LIN {X 0,Y 405.489,Z 1080.281,A -85,B 0,C 180,E1 13917.147,E2 13917.147} C_VEL
LIN {X 0,Y 408.998,Z 1063.709,A -85,B 0,C 180,E1 13914.736,E2 13914.736} C_VEL
LIN {X 0,Y 412.817,Z 1045.417,A -85,B 0,C 180,E1 13912.472,E2 13912.472} C_VEL
LIN {X 0,Y 416.994,Z 1024.781,A -85,B 0,C 180,E1 13910.291,E2 13910.291} C_VEL
LIN {X 0,Y 420.9,Z 1004.657,A -85,B 0,C 180,E1 13908.488,E2 13908.488} C_VEL
LIN {X 0,Y 424.408,Z 984.623,A -85,B 0,C 180,E1 13906.997,E2 13906.997} C_VEL
LIN {X 0,Y 427.831,Z 963.376,A -85,B 0,C 180,E1 13905.671,E2 13905.671} C_VEL
LIN {X 0,Y 430.64,Z 942.779,A -85,B 0,C 180,E1 13904.632,E2 13904.632} C_VEL
LIN {X 0,Y 433.258,Z 920.08,A -85,B 0,C 180,E1 13903.723,E2 13903.723} C_VEL
LIN {X 0,Y 435.218,Z 898.048,A -85,B 0,C 180,E1 13903.072,E2 13903.072} C_VEL
LIN {X 0,Y 436.86,Z 866.302,A -85,B 0,C 180,E1 13902.413,E2 13902.413} C_VEL
LIN {X 0,Y 445.415,Z 656.553,A -85,B 0,C 180,E1 13898.433,E2 13898.433} C_VEL
LIN {X 0,Y 447.125,Z 611.826,A -85,B 0,C 180,E1 13897.563,E2 13897.563} C_VEL
LIN {X 0,Y 435.207,Z 593.667,A -85,B 0,C 180,E1 13895.175,E2 13895.175} C_VEL
LIN {X 0,Y 424.65,Z 578.968,A -85,B 0,C 180,E1 13892.869,E2 13892.869} C_VEL
LIN {X 0,Y 417.413,Z 569.477,A -85,B 0,C 180,E1 13891.157,E2 13891.157} C_VEL
LIN {X 0,Y 413.791,Z 564.844,A -85,B 0,C 180,E1 13890.252,E2 13890.252} C_VEL
LIN {X 0,Y 409.785,Z 559.833,A -85,B 0,C 180,E1 13889.208,E2 13889.208} C_VEL
LIN {X 0,Y 405.456,Z 554.439,A -85,B 0,C 180,E1 13887.999,E2 13887.999} C_VEL
LIN {X 0,Y 402.661,Z 549.627,A -85,B 0,C 180,E1 13886.548,E2 13886.548} C_VEL
LIN {X 0,Y 400.386,Z 545.696,A -85,B 0,C 180,E1 13885.279,E2 13885.279} C_VEL
LIN {X 0,Y 397.379,Z 541.061,A -85,B 0,C 180,E1 13883.582,E2 13883.582} C_VEL
LIN {X 0,Y 396.535,Z 539.345,A -85,B 0,C 180,E1 13883.006,E2 13883.006} C_VEL
LIN {X 0,Y 394.114,Z 536.079,A -85,B 0,C 180,E1 13881.583,E2 13881.583} C_VEL
LIN {X 0,Y 393.583,Z 534.195,A -85,B 0,C 180,E1 13880.833,E2 13880.833} C_VEL
LIN {X 0,Y 393.553,Z 533.972,A -85,B 0,C 180,E1 13876.835,E2 13876.835} C_VEL
LIN {X 0,Y 393.555,Z 533.997,A -85,B 0,C 180,E1 13872.918,E2 13872.918} C_VEL
LIN {X 0,Y 393.548,Z 533.952,A -85,B 0,C 180,E1 13868.915,E2 13868.915} C_VEL
LIN {X 0,Y 393.557,Z 534.026,A -85,B 0,C 180,E1 13864.955,E2 13864.955} C_VEL
LIN {X 0,Y 393.56,Z 534.017,A -85,B 0,C 180,E1 13860.873,E2 13860.873} C_VEL
LIN {X 0,Y 393.555,Z 534.013,A -85,B 0,C 180,E1 13856.941,E2 13856.941} C_VEL
LIN {X 0,Y 393.549,Z 534.009,A -85,B 0,C 180,E1 13852.995,E2 13852.995} C_VEL
LIN {X 0,Y 393.543,Z 533.975,A -85,B 0,C 180,E1 13849.015,E2 13849.015} C_VEL
LIN {X 0,Y 393.55,Z 533.997,A -85,B 0,C 180,E1 13844.98,E2 13844.98} C_VEL
LIN {X 0,Y 393.552,Z 533.958,A -85,B 0,C 180,E1 13841.022,E2 13841.022} C_VEL
LIN {X 0,Y 393.573,Z 534.093,A -85,B 0,C 180,E1 13836.968,E2 13836.968} C_VEL
LIN {X 0,Y 393.64,Z 534.566,A -85,B 0,C 180,E1 13836.485,E2 13836.485} C_VEL
LIN {X 0,Y 395.297,Z 538.039,A -85,B 0,C 180,E1 13835.173,E2 13835.173} C_VEL
LIN {X 0,Y 396.887,Z 539.799,A -85,B 0,C 180,E1 13834.322,E2 13834.322} C_VEL
LIN {X 0,Y 398.83,Z 543.682,A -85,B 0,C 180,E1 13833.014,E2 13833.014} C_VEL
LIN {X 0,Y 400.178,Z 545.463,A -85,B 0,C 180,E1 13832.307,E2 13832.307} C_VEL
LIN {X 0,Y 402.489,Z 549.53,A -85,B 0,C 180,E1 13830.979,E2 13830.979} C_VEL
LIN {X 0,Y 406.12,Z 555.885,A -85,B 0,C 180,E1 13829.032,E2 13829.032} C_VEL
LIN {X 0,Y 411.461,Z 565.678,A -85,B 0,C 180,E1 13826.355,E2 13826.355} C_VEL
LIN {X 0,Y 417.794,Z 577.852,A -85,B 0,C 180,E1 13823.423,E2 13823.423} C_VEL
LIN {X 0,Y 419.708,Z 581.207,A -85,B 0,C 180,E1 13822.764,E2 13822.764} C_VEL
LIN {X 0,Y 431.985,Z 599.336,A -85,B 0,C 180,E1 13819.994,E2 13819.994} C_VEL
LIN {X 0,Y 441.06,Z 613.989,A -85,B 0,C 180,E1 13818.116,E2 13818.116} C_VEL
LIN {X 0,Y 443.278,Z 632.103,A -85,B 0,C 180,E1 13817.332,E2 13817.332} C_VEL
LIN {X 0,Y 435.43,Z 864.5,A -85,B 0,C 180,E1 13813.233,E2 13813.233} C_VEL
LIN {X 0,Y 434.04,Z 899.876,A -85,B 0,C 180,E1 13812.574,E2 13812.574} C_VEL
LIN {X 0,Y 432.284,Z 921.112,A -85,B 0,C 180,E1 13811.981,E2 13811.981} C_VEL
LIN {X 0,Y 429.933,Z 942.214,A -85,B 0,C 180,E1 13811.159,E2 13811.159} C_VEL
LIN {X 0,Y 427.165,Z 962.307,A -85,B 0,C 180,E1 13810.155,E2 13810.155} C_VEL
LIN {X 0,Y 423.94,Z 981.509,A -85,B 0,C 180,E1 13808.943,E2 13808.943} C_VEL
LIN {X 0,Y 420.069,Z 1001.923,A -85,B 0,C 180,E1 13807.37,E2 13807.37} C_VEL
LIN {X 0,Y 418.412,Z 1010.233,A -85,B 0,C 180,E1 13806.635,E2 13806.635} C_VEL
LIN {X 0,Y 416.201,Z 1016.718,A -85,B 0,C 180,E1 13806.1,E2 13806.1} C_VEL
LIN {X 0,Y 407.722,Z 1032.836,A -85,B 0,C 180,E1 13804.905,E2 13804.905} C_VEL
LIN {X 0,Y 405.499,Z 1038.649,A -85,B 0,C 180,E1 13804.288,E2 13804.288} C_VEL
LIN {X 0,Y 401.382,Z 1055.192,A -85,B 0,C 180,E1 13802.046,E2 13802.046} C_VEL
LIN {X 0,Y 397.658,Z 1069.963,A -85,B 0,C 180,E1 13799.692,E2 13799.692} C_VEL
LIN {X 0,Y 394.167,Z 1083.713,A -85,B 0,C 180,E1 13797.081,E2 13797.081} C_VEL
LIN {X 0,Y 391.006,Z 1096.711,A -85,B 0,C 180,E1 13794.151,E2 13794.151} C_VEL
LIN {X 0,Y 388.496,Z 1107.96,A -85,B 0,C 180,E1 13791.12,E2 13791.12} C_VEL
LIN {X 0,Y 386.647,Z 1117.265,A -85,B 0,C 180,E1 13788.078,E2 13788.078} C_VEL
LIN {X 0,Y 385.339,Z 1125.185,A -85,B 0,C 180,E1 13784.885,E2 13784.885} C_VEL
LIN {X 0,Y 384.562,Z 1131.485,A -85,B 0,C 180,E1 13781.701,E2 13781.701} C_VEL
LIN {X 0,Y 384.149,Z 1136.202,A -85,B 0,C 180,E1 13778.481,E2 13778.481} C_VEL
LIN {X 0,Y 383.963,Z 1139.441,A -85,B 0,C 180,E1 13775.229,E2 13775.229} C_VEL
LIN {X 0,Y 383.933,Z 1141.104,A -85,B 0,C 180,E1 13772.239,E2 13772.239} C_VEL
LIN {X 0,Y 383.927,Z 1141.391,A -85,B 0,C 180,E1 13769.105,E2 13769.105} C_VEL
LIN {X 0,Y 383.954,Z 1140.362,A -85,B 0,C 180,E1 13765.968,E2 13765.968} C_VEL
LIN {X 0,Y 384.043,Z 1137.764,A -85,B 0,C 180,E1 13762.821,E2 13762.821} C_VEL
LIN {X 0,Y 384.341,Z 1133.558,A -85,B 0,C 180,E1 13759.508,E2 13759.508} C_VEL
LIN {X 0,Y 384.971,Z 1127.979,A -85,B 0,C 180,E1 13756.329,E2 13756.329} C_VEL
LIN {X 0,Y 386.05,Z 1120.698,A -85,B 0,C 180,E1 13753.137,E2 13753.137} C_VEL
LIN {X 0,Y 387.723,Z 1111.688,A -85,B 0,C 180,E1 13749.941,E2 13749.941} C_VEL
LIN {X 0,Y 389.978,Z 1101.243,A -85,B 0,C 180,E1 13746.904,E2 13746.904} C_VEL
LIN {X 0,Y 392.768,Z 1089.341,A -85,B 0,C 180,E1 13744.033,E2 13744.033} C_VEL
LIN {X 0,Y 396.279,Z 1075.322,A -85,B 0,C 180,E1 13741.189,E2 13741.189} C_VEL
LIN {X 0,Y 400.044,Z 1060.64,A -85,B 0,C 180,E1 13738.676,E2 13738.676} C_VEL
LIN {X 0,Y 403.981,Z 1044.856,A -85,B 0,C 180,E1 13736.416,E2 13736.416} C_VEL
LIN {X 0,Y 408.286,Z 1027.046,A -85,B 0,C 180,E1 13734.263,E2 13734.263} C_VEL
LIN {X 0,Y 412.346,Z 1009.31,A -85,B 0,C 180,E1 13732.459,E2 13732.459} C_VEL
LIN {X 0,Y 416.157,Z 990.732,A -85,B 0,C 180,E1 13730.9,E2 13730.9} C_VEL
LIN {X 0,Y 419.96,Z 969.91,A -85,B 0,C 180,E1 13729.46,E2 13729.46} C_VEL
LIN {X 0,Y 423.147,Z 949.876,A -85,B 0,C 180,E1 13728.346,E2 13728.346} C_VEL
LIN {X 0,Y 425.704,Z 929.539,A -85,B 0,C 180,E1 13727.472,E2 13727.472} C_VEL
LIN {X 0,Y 427.863,Z 907.472,A -85,B 0,C 180,E1 13726.765,E2 13726.765} C_VEL
LIN {X 0,Y 429.218,Z 885.36,A -85,B 0,C 180,E1 13726.277,E2 13726.277} C_VEL
LIN {X 0,Y 437.154,Z 658.958,A -85,B 0,C 180,E1 13722.256,E2 13722.256} C_VEL
LIN {X 0,Y 437.807,Z 637.947,A -85,B 0,C 180,E1 13721.847,E2 13721.847} C_VEL
LIN {X 0,Y 434.549,Z 619.163,A -85,B 0,C 180,E1 13720.847,E2 13720.847} C_VEL
LIN {X 0,Y 428.925,Z 610.299,A -85,B 0,C 180,E1 13719.653,E2 13719.653} C_VEL
LIN {X 0,Y 424.479,Z 614.666,A -85,B 0,C 180,E1 13718.971,E2 13718.971} C_VEL
LIN {X 0,Y 422.787,Z 616.084,A -85,B 0,C 180,E1 13718.697,E2 13718.697} C_VEL
LIN {X 0,Y 418.036,Z 623.156,A -85,B 0,C 180,E1 13717.995,E2 13717.995} C_VEL
LIN {X 0,Y 414.316,Z 626.731,A -85,B 0,C 180,E1 13717.369,E2 13717.369} C_VEL
LIN {X 0,Y 412.783,Z 627.888,A -85,B 0,C 180,E1 13717.095,E2 13717.095} C_VEL
LIN {X 0,Y 408.266,Z 635.452,A -85,B 0,C 180,E1 13716.39,E2 13716.39} C_VEL
LIN {X 0,Y 405.178,Z 638.802,A -85,B 0,C 180,E1 13715.836,E2 13715.836} C_VEL
LIN {X 0,Y 403.521,Z 640.351,A -85,B 0,C 180,E1 13715.414,E2 13715.414} C_VEL
LIN {X 0,Y 402.905,Z 644.108,A -85,B 0,C 180,E1 13714.978,E2 13714.978} C_VEL
LIN {X 0,Y 400.433,Z 687.457,A -85,B 0,C 180,E1 13711.123,E2 13711.123} C_VEL
LIN {X 0,Y 398.504,Z 724.534,A -85,B 0,C 180,E1 13707.877,E2 13707.877} C_VEL
LIN {X 0,Y 399.176,Z 732.919,A -85,B 0,C 180,E1 13707.639,E2 13707.639} C_VEL
LIN {X 0,Y 394.985,Z 896.313,A -85,B 0,C 180,E1 13704.201,E2 13704.201} C_VEL
LIN {X 0,Y 394.483,Z 914.11,A -85,B 0,C 180,E1 13703.563,E2 13703.563} C_VEL
LIN {X 0,Y 393.686,Z 931.61,A -85,B 0,C 180,E1 13702.657,E2 13702.657} C_VEL
LIN {X 0,Y 392.701,Z 948.326,A -85,B 0,C 180,E1 13701.509,E2 13701.509} C_VEL
LIN {X 0,Y 391.593,Z 963.531,A -85,B 0,C 180,E1 13700.164,E2 13700.164} C_VEL
LIN {X 0,Y 390.381,Z 978.468,A -85,B 0,C 180,E1 13698.518,E2 13698.518} C_VEL
LIN {X 0,Y 389.222,Z 991.674,A -85,B 0,C 180,E1 13696.721,E2 13696.721} C_VEL
LIN {X 0,Y 388.165,Z 1003.238,A -85,B 0,C 180,E1 13694.775,E2 13694.775} C_VEL
LIN {X 0,Y 387.252,Z 1013.798,A -85,B 0,C 180,E1 13692.584,E2 13692.584} C_VEL
LIN {X 0,Y 386.584,Z 1022.094,A -85,B 0,C 180,E1 13690.431,E2 13690.431} C_VEL
LIN {X 0,Y 386.073,Z 1029.198,A -85,B 0,C 180,E1 13688.04,E2 13688.04} C_VEL
LIN {X 0,Y 385.793,Z 1034.56,A -85,B 0,C 180,E1 13685.605,E2 13685.605} C_VEL
LIN {X 0,Y 385.689,Z 1038.235,A -85,B 0,C 180,E1 13683.121,E2 13683.121} C_VEL
LIN {X 0,Y 385.709,Z 1040.12,A -85,B 0,C 180,E1 13680.595,E2 13680.595} C_VEL
LIN {X 0,Y 385.833,Z 1040.274,A -85,B 0,C 180,E1 13678.07,E2 13678.07} C_VEL
LIN {X 0,Y 386.089,Z 1038.661,A -85,B 0,C 180,E1 13675.545,E2 13675.545} C_VEL
LIN {X 0,Y 386.474,Z 1035.386,A -85,B 0,C 180,E1 13673.166,E2 13673.166} C_VEL
LIN {X 0,Y 387.055,Z 1030.333,A -85,B 0,C 180,E1 13670.784,E2 13670.784} C_VEL
LIN {X 0,Y 387.872,Z 1023.313,A -85,B 0,C 180,E1 13668.399,E2 13668.399} C_VEL
LIN {X 0,Y 388.76,Z 1015.216,A -85,B 0,C 180,E1 13666.314,E2 13666.314} C_VEL
LIN {X 0,Y 389.856,Z 1004.907,A -85,B 0,C 180,E1 13664.226,E2 13664.226} C_VEL
LIN {X 0,Y 391.015,Z 993.39,A -85,B 0,C 180,E1 13662.362,E2 13662.362} C_VEL
LIN {X 0,Y 392.13,Z 980.673,A -85,B 0,C 180,E1 13660.72,E2 13660.72} C_VEL
LIN {X 0,Y 393.185,Z 966.201,A -85,B 0,C 180,E1 13659.225,E2 13659.225} C_VEL
LIN {X 0,Y 394.052,Z 951.531,A -85,B 0,C 180,E1 13658.022,E2 13658.022} C_VEL
LIN {X 0,Y 394.739,Z 935.274,A -85,B 0,C 180,E1 13657.002,E2 13657.002} C_VEL
LIN {X 0,Y 395.201,Z 917.715,A -85,B 0,C 180,E1 13656.196,E2 13656.196} C_VEL
LIN {X 0,Y 395.358,Z 898.366,A -85,B 0,C 180,E1 13655.623,E2 13655.623} C_VEL
LIN {X 0,Y 397.596,Z 820.71,A -85,B 0,C 180,E1 13653.836,E2 13653.836} C_VEL
LIN {X 0,Y 401.124,Z 744.737,A -85,B 0,C 180,E1 13651.935,E2 13651.935} C_VEL
LIN {X 0,Y 403.455,Z 734.084,A -85,B 0,C 180,E1 13651.264,E2 13651.264} C_VEL
LIN {X 0,Y 405.647,Z 691.359,A -85,B 0,C 180,E1 13647.665,E2 13647.665} C_VEL
LIN {X 0,Y 406.635,Z 689.08,A -85,B 0,C 180,E1 13647.336,E2 13647.336} C_VEL
LIN {X 0,Y 409.817,Z 685.698,A -85,B 0,C 180,E1 13646.799,E2 13646.799} C_VEL
LIN {X 0,Y 414.057,Z 678.624,A -85,B 0,C 180,E1 13646.2,E2 13646.2} C_VEL
LIN {X 0,Y 415.402,Z 676.435,A -85,B 0,C 180,E1 13646.013,E2 13646.013} C_VEL
LIN {X 0,Y 419.171,Z 672.646,A -85,B 0,C 180,E1 13645.431,E2 13645.431} C_VEL
LIN {X 0,Y 423.613,Z 665.769,A -85,B 0,C 180,E1 13644.837,E2 13644.837} C_VEL
LIN {X 0,Y 424.895,Z 663.76,A -85,B 0,C 180,E1 13644.67,E2 13644.67} C_VEL
LIN {X 0,Y 429.408,Z 659.017,A -85,B 0,C 180,E1 13644.031,E2 13644.031} C_VEL
LIN {X 0,Y 434.063,Z 651.878,A -85,B 0,C 180,E1 13643.456,E2 13643.456} C_VEL
LIN {X 0,Y 440.003,Z 645.272,A -85,B 0,C 180,E1 13642.684,E2 13642.684} C_VEL
LIN {X 0,Y 440.743,Z 644.394,A -85,B 0,C 180,E1 13642.592,E2 13642.592} C_VEL
LIN {X 0,Y 431.895,Z 850.784,A -85,B 0,C 180,E1 13638.641,E2 13638.641} C_VEL
LIN {X 0,Y 429.828,Z 894.793,A -85,B 0,C 180,E1 13637.764,E2 13637.764} C_VEL
LIN {X 0,Y 427.715,Z 917.794,A -85,B 0,C 180,E1 13637.103,E2 13637.103} C_VEL
LIN {X 0,Y 424.904,Z 941.779,A -85,B 0,C 180,E1 13636.157,E2 13636.157} C_VEL
LIN {X 0,Y 421.963,Z 962.479,A -85,B 0,C 180,E1 13635.113,E2 13635.113} C_VEL
LIN {X 0,Y 418.395,Z 983.875,A -85,B 0,C 180,E1 13633.776,E2 13633.776} C_VEL
LIN {X 0,Y 414.643,Z 1004.331,A -85,B 0,C 180,E1 13632.245,E2 13632.245} C_VEL
LIN {X 0,Y 410.61,Z 1024.083,A -85,B 0,C 180,E1 13630.462,E2 13630.462} C_VEL
LIN {X 0,Y 406.335,Z 1044.207,A -85,B 0,C 180,E1 13628.323,E2 13628.323} C_VEL
LIN {X 0,Y 402.487,Z 1061.551,A -85,B 0,C 180,E1 13626.162,E2 13626.162} C_VEL
LIN {X 0,Y 398.547,Z 1079.124,A -85,B 0,C 180,E1 13623.602,E2 13623.602} C_VEL
LIN {X 0,Y 395.061,Z 1095.078,A -85,B 0,C 180,E1 13620.911,E2 13620.911} C_VEL
LIN {X 0,Y 392.014,Z 1109.49,A -85,B 0,C 180,E1 13618.056,E2 13618.056} C_VEL
LIN {X 0,Y 389.359,Z 1123.169,A -85,B 0,C 180,E1 13614.907,E2 13614.907} C_VEL
LIN {X 0,Y 387.555,Z 1133.447,A -85,B 0,C 180,E1 13612.128,E2 13612.128} C_VEL
LIN {X 0,Y 386.011,Z 1143.518,A -85,B 0,C 180,E1 13608.892,E2 13608.892} C_VEL
LIN {X 0,Y 385.06,Z 1151.04,A -85,B 0,C 180,E1 13605.977,E2 13605.977} C_VEL
LIN {X 0,Y 384.384,Z 1158.01,A -85,B 0,C 180,E1 13602.621,E2 13602.621} C_VEL
LIN {X 0,Y 384.075,Z 1162.606,A -85,B 0,C 180,E1 13599.742,E2 13599.742} C_VEL
LIN {X 0,Y 383.951,Z 1166.356,A -85,B 0,C 180,E1 13596.58,E2 13596.58} C_VEL
LIN {X 0,Y 383.899,Z 1168.515,A -85,B 0,C 180,E1 13593.434,E2 13593.434} C_VEL
LIN {X 0,Y 383.898,Z 1169.345,A -85,B 0,C 180,E1 13590.597,E2 13590.597} C_VEL
LIN {X 0,Y 383.907,Z 1168.869,A -85,B 0,C 180,E1 13587.313,E2 13587.313} C_VEL
LIN {X 0,Y 383.92,Z 1167.184,A -85,B 0,C 180,E1 13584.47,E2 13584.47} C_VEL
LIN {X 0,Y 384.031,Z 1164.056,A -85,B 0,C 180,E1 13581.315,E2 13581.315} C_VEL
LIN {X 0,Y 384.301,Z 1159.143,A -85,B 0,C 180,E1 13578.028,E2 13578.028} C_VEL
LIN {X 0,Y 384.829,Z 1153.157,A -85,B 0,C 180,E1 13574.941,E2 13574.941} C_VEL
LIN {X 0,Y 385.834,Z 1144.804,A -85,B 0,C 180,E1 13571.569,E2 13571.569} C_VEL
LIN {X 0,Y 387.224,Z 1135.587,A -85,B 0,C 180,E1 13568.49,E2 13568.49} C_VEL
LIN {X 0,Y 389.14,Z 1124.397,A -85,B 0,C 180,E1 13565.402,E2 13565.402} C_VEL
LIN {X 0,Y 391.621,Z 1111.508,A -85,B 0,C 180,E1 13562.366,E2 13562.366} C_VEL
LIN {X 0,Y 394.579,Z 1097.191,A -85,B 0,C 180,E1 13559.491,E2 13559.491} C_VEL
LIN {X 0,Y 398.211,Z 1080.656,A -85,B 0,C 180,E1 13556.641,E2 13556.641} C_VEL
LIN {X 0,Y 401.9,Z 1064.246,A -85,B 0,C 180,E1 13554.196,E2 13554.196} C_VEL
LIN {X 0,Y 405.91,Z 1046.072,A -85,B 0,C 180,E1 13551.899,E2 13551.899} C_VEL
LIN {X 0,Y 410.149,Z 1026.318,A -85,B 0,C 180,E1 13549.758,E2 13549.758} C_VEL
LIN {X 0,Y 414.009,Z 1007.308,A -85,B 0,C 180,E1 13548.012,E2 13548.012} C_VEL
LIN {X 0,Y 418.021,Z 985.885,A -85,B 0,C 180,E1 13546.365,E2 13546.365} C_VEL
LIN {X 0,Y 421.587,Z 964.983,A -85,B 0,C 180,E1 13545.028,E2 13545.028} C_VEL
LIN {X 0,Y 424.699,Z 943.196,A -85,B 0,C 180,E1 13543.911,E2 13543.911} C_VEL
LIN {X 0,Y 427.414,Z 920.823,A -85,B 0,C 180,E1 13543.002,E2 13543.002} C_VEL
LIN {X 0,Y 429.472,Z 898.652,A -85,B 0,C 180,E1 13542.339,E2 13542.339} C_VEL
LIN {X 0,Y 431.189,Z 867.354,A -85,B 0,C 180,E1 13541.679,E2 13541.679} C_VEL
LIN {X 0,Y 440.129,Z 657.984,A -85,B 0,C 180,E1 13537.672,E2 13537.672} C_VEL
LIN {X 0,Y 441.842,Z 615.744,A -85,B 0,C 180,E1 13536.846,E2 13536.846} C_VEL
LIN {X 0,Y 430.859,Z 598.912,A -85,B 0,C 180,E1 13534.568,E2 13534.568} C_VEL
LIN {X 0,Y 419.745,Z 583.174,A -85,B 0,C 180,E1 13532.046,E2 13532.046} C_VEL
LIN {X 0,Y 410.765,Z 571.557,A -85,B 0,C 180,E1 13529.813,E2 13529.813} C_VEL
LIN {X 0,Y 406.699,Z 566.451,A -85,B 0,C 180,E1 13528.726,E2 13528.726} C_VEL
LIN {X 0,Y 402.422,Z 561.153,A -85,B 0,C 180,E1 13527.524,E2 13527.524} C_VEL
LIN {X 0,Y 397.873,Z 555.704,A -85,B 0,C 180,E1 13526.169,E2 13526.169} C_VEL
LIN {X 0,Y 395.181,Z 551.082,A -85,B 0,C 180,E1 13524.675,E2 13524.675} C_VEL
LIN {X 0,Y 392.967,Z 547.647,A -85,B 0,C 180,E1 13523.385,E2 13523.385} C_VEL
LIN {X 0,Y 392.14,Z 545.932,A -85,B 0,C 180,E1 13522.802,E2 13522.802} C_VEL
LIN {X 0,Y 389.596,Z 542.202,A -85,B 0,C 180,E1 13521.214,E2 13521.214} C_VEL
LIN {X 0,Y 388.881,Z 540.571,A -85,B 0,C 180,E1 13520.624,E2 13520.624} C_VEL
LIN {X 0,Y 386.225,Z 537.218,A -85,B 0,C 180,E1 13518.88,E2 13518.88} C_VEL
LIN {X 0,Y 385.644,Z 535.176,A -85,B 0,C 180,E1 13517.97,E2 13517.97} C_VEL
LIN {X 0,Y 385.609,Z 534.952,A -85,B 0,C 180,E1 13514.107,E2 13514.107} C_VEL
LIN {X 0,Y 385.608,Z 534.955,A -85,B 0,C 180,E1 13510.155,E2 13510.155} C_VEL
LIN {X 0,Y 385.615,Z 534.984,A -85,B 0,C 180,E1 13506.102,E2 13506.102} C_VEL
LIN {X 0,Y 385.618,Z 535.007,A -85,B 0,C 180,E1 13502.08,E2 13502.08} C_VEL
LIN {X 0,Y 385.62,Z 535.014,A -85,B 0,C 180,E1 13498.068,E2 13498.068} C_VEL
LIN {X 0,Y 385.62,Z 535.01,A -85,B 0,C 180,E1 13494.047,E2 13494.047} C_VEL
LIN {X 0,Y 385.617,Z 534.99,A -85,B 0,C 180,E1 13489.995,E2 13489.995} C_VEL
LIN {X 0,Y 385.614,Z 534.956,A -85,B 0,C 180,E1 13485.871,E2 13485.871} C_VEL
LIN {X 0,Y 385.617,Z 534.953,A -85,B 0,C 180,E1 13481.871,E2 13481.871} C_VEL
LIN {X 0,Y 385.655,Z 535.233,A -85,B 0,C 180,E1 13479.512,E2 13479.512} C_VEL
LIN {X 0,Y 387.264,Z 538.949,A -85,B 0,C 180,E1 13477.855,E2 13477.855} C_VEL
LIN {X 0,Y 389.132,Z 541.095,A -85,B 0,C 180,E1 13476.69,E2 13476.69} C_VEL
LIN {X 0,Y 391.146,Z 544.903,A -85,B 0,C 180,E1 13475.214,E2 13475.214} C_VEL
LIN {X 0,Y 392.596,Z 546.938,A -85,B 0,C 180,E1 13474.345,E2 13474.345} C_VEL
LIN {X 0,Y 394.94,Z 550.888,A -85,B 0,C 180,E1 13472.89,E2 13472.89} C_VEL
LIN {X 0,Y 398.658,Z 557.383,A -85,B 0,C 180,E1 13470.72,E2 13470.72} C_VEL
LIN {X 0,Y 401.534,Z 562.592,A -85,B 0,C 180,E1 13469.138,E2 13469.138} C_VEL
LIN {X 0,Y 406.295,Z 571.246,A -85,B 0,C 180,E1 13466.716,E2 13466.716} C_VEL
LIN {X 0,Y 410.836,Z 579.749,A -85,B 0,C 180,E1 13464.646,E2 13464.646} C_VEL
LIN {X 0,Y 421.537,Z 595.199,A -85,B 0,C 180,E1 13462.01,E2 13462.01} C_VEL
LIN {X 0,Y 431.227,Z 610.153,A -85,B 0,C 180,E1 13459.844,E2 13459.844} C_VEL
LIN {X 0,Y 436.351,Z 618.754,A -85,B 0,C 180,E1 13458.76,E2 13458.76} C_VEL
LIN {X 0,Y 438.095,Z 633.737,A -85,B 0,C 180,E1 13458.106,E2 13458.106} C_VEL
LIN {X 0,Y 429.791,Z 866.944,A -85,B 0,C 180,E1 13453.956,E2 13453.956} C_VEL
LIN {X 0,Y 428.382,Z 900.23,A -85,B 0,C 180,E1 13453.325,E2 13453.325} C_VEL
LIN {X 0,Y 426.554,Z 921.396,A -85,B 0,C 180,E1 13452.729,E2 13452.729} C_VEL
LIN {X 0,Y 424.09,Z 942.521,A -85,B 0,C 180,E1 13451.898,E2 13451.898} C_VEL
LIN {X 0,Y 421.305,Z 961.97,A -85,B 0,C 180,E1 13450.921,E2 13450.921} C_VEL
LIN {X 0,Y 417.937,Z 981.261,A -85,B 0,C 180,E1 13449.7,E2 13449.7} C_VEL
LIN {X 0,Y 414.058,Z 1000.959,A -85,B 0,C 180,E1 13448.184,E2 13448.184} C_VEL
LIN {X 0,Y 410.151,Z 1019.023,A -85,B 0,C 180,E1 13446.5,E2 13446.5} C_VEL
LIN {X 0,Y 406.081,Z 1036.243,A -85,B 0,C 180,E1 13444.579,E2 13444.579} C_VEL
LIN {X 0,Y 405.499,Z 1038.649,A -85,B 0,C 180,E1 13444.288,E2 13444.288} C_VEL
LIN {X 0,Y 403.25,Z 1044.503,A -85,B 0,C 180,E1 13443.637,E2 13443.637} C_VEL
LIN {X 0,Y 394.465,Z 1059.022,A -85,B 0,C 180,E1 13442.081,E2 13442.081} C_VEL
LIN {X 0,Y 392.203,Z 1064.271,A -85,B 0,C 180,E1 13441.32,E2 13441.32} C_VEL
LIN {X 0,Y 388.422,Z 1078.535,A -85,B 0,C 180,E1 13438.775,E2 13438.775} C_VEL
LIN {X 0,Y 384.999,Z 1091.419,A -85,B 0,C 180,E1 13436.028,E2 13436.028} C_VEL
LIN {X 0,Y 381.986,Z 1103.523,A -85,B 0,C 180,E1 13432.955,E2 13432.955} C_VEL
LIN {X 0,Y 379.709,Z 1113.699,A -85,B 0,C 180,E1 13429.858,E2 13429.858} C_VEL
LIN {X 0,Y 378.083,Z 1122.002,A -85,B 0,C 180,E1 13426.754,E2 13426.754} C_VEL
LIN {X 0,Y 376.934,Z 1129.317,A -85,B 0,C 180,E1 13423.343,E2 13423.343} C_VEL
LIN {X 0,Y 376.326,Z 1134.709,A -85,B 0,C 180,E1 13420.099,E2 13420.099} C_VEL
LIN {X 0,Y 376.057,Z 1138.451,A -85,B 0,C 180,E1 13416.872,E2 13416.872} C_VEL
LIN {X 0,Y 375.948,Z 1140.882,A -85,B 0,C 180,E1 13413.507,E2 13413.507} C_VEL
LIN {X 0,Y 375.93,Z 1141.735,A -85,B 0,C 180,E1 13410.457,E2 13410.457} C_VEL
LIN {X 0,Y 375.935,Z 1141.179,A -85,B 0,C 180,E1 13407.103,E2 13407.103} C_VEL
LIN {X 0,Y 376.018,Z 1139.274,A -85,B 0,C 180,E1 13403.894,E2 13403.894} C_VEL
LIN {X 0,Y 376.234,Z 1135.802,A -85,B 0,C 180,E1 13400.671,E2 13400.671} C_VEL
LIN {X 0,Y 376.764,Z 1130.638,A -85,B 0,C 180,E1 13397.275,E2 13397.275} C_VEL
LIN {X 0,Y 377.675,Z 1124.4,A -85,B 0,C 180,E1 13394.176,E2 13394.176} C_VEL
LIN {X 0,Y 379.191,Z 1116.138,A -85,B 0,C 180,E1 13390.915,E2 13390.915} C_VEL
LIN {X 0,Y 381.338,Z 1106.365,A -85,B 0,C 180,E1 13387.753,E2 13387.753} C_VEL
LIN {X 0,Y 384.098,Z 1095.012,A -85,B 0,C 180,E1 13384.728,E2 13384.728} C_VEL
LIN {X 0,Y 387.291,Z 1082.668,A -85,B 0,C 180,E1 13381.974,E2 13381.974} C_VEL
LIN {X 0,Y 390.939,Z 1069.16,A -85,B 0,C 180,E1 13379.405,E2 13379.405} C_VEL
LIN {X 0,Y 394.901,Z 1054.226,A -85,B 0,C 180,E1 13377.019,E2 13377.019} C_VEL
LIN {X 0,Y 399.146,Z 1037.989,A -85,B 0,C 180,E1 13374.82,E2 13374.82} C_VEL
LIN {X 0,Y 403.351,Z 1021.168,A -85,B 0,C 180,E1 13372.888,E2 13372.888} C_VEL
LIN {X 0,Y 407.426,Z 1003.213,A -85,B 0,C 180,E1 13371.169,E2 13371.169} C_VEL
LIN {X 0,Y 411.643,Z 983.021,A -85,B 0,C 180,E1 13369.569,E2 13369.569} C_VEL
LIN {X 0,Y 415.132,Z 963.978,A -85,B 0,C 180,E1 13368.336,E2 13368.336} C_VEL
LIN {X 0,Y 418.235,Z 943.606,A -85,B 0,C 180,E1 13367.285,E2 13367.285} C_VEL
LIN {X 0,Y 420.798,Z 923.048,A -85,B 0,C 180,E1 13366.455,E2 13366.455} C_VEL
LIN {X 0,Y 422.741,Z 901.646,A -85,B 0,C 180,E1 13365.837,E2 13365.837} C_VEL
LIN {X 0,Y 424.172,Z 871.612,A -85,B 0,C 180,E1 13365.249,E2 13365.249} C_VEL
LIN {X 0,Y 432.502,Z 648.361,A -85,B 0,C 180,E1 13361.242,E2 13361.242} C_VEL
LIN {X 0,Y 432.699,Z 639.79,A -85,B 0,C 180,E1 13361.059,E2 13361.059} C_VEL
LIN {X 0,Y 430.033,Z 623.992,A -85,B 0,C 180,E1 13360.203,E2 13360.203} C_VEL
LIN {X 0,Y 427.706,Z 620.326,A -85,B 0,C 180,E1 13359.701,E2 13359.701} C_VEL
LIN {X 0,Y 425.003,Z 622.739,A -85,B 0,C 180,E1 13359.283,E2 13359.283} C_VEL
LIN {X 0,Y 420.137,Z 629.624,A -85,B 0,C 180,E1 13358.574,E2 13358.574} C_VEL
LIN {X 0,Y 415.812,Z 633.76,A -85,B 0,C 180,E1 13357.863,E2 13357.863} C_VEL
LIN {X 0,Y 414.768,Z 634.887,A -85,B 0,C 180,E1 13357.691,E2 13357.691} C_VEL
LIN {X 0,Y 410.166,Z 642.057,A -85,B 0,C 180,E1 13356.978,E2 13356.978} C_VEL
LIN {X 0,Y 406.429,Z 645.936,A -85,B 0,C 180,E1 13356.319,E2 13356.319} C_VEL
LIN {X 0,Y 404.774,Z 647.302,A -85,B 0,C 180,E1 13356.008,E2 13356.008} C_VEL
LIN {X 0,Y 400.09,Z 655.519,A -85,B 0,C 180,E1 13355.239,E2 13355.239} C_VEL
LIN {X 0,Y 396.99,Z 659.125,A -85,B 0,C 180,E1 13354.651,E2 13354.651} C_VEL
LIN {X 0,Y 395.3,Z 660.873,A -85,B 0,C 180,E1 13354.197,E2 13354.197} C_VEL
LIN {X 0,Y 394.74,Z 664.359,A -85,B 0,C 180,E1 13353.788,E2 13353.788} C_VEL
LIN {X 0,Y 391.964,Z 710.415,A -85,B 0,C 180,E1 13349.662,E2 13349.662} C_VEL
LIN {X 0,Y 391.239,Z 725.392,A -85,B 0,C 180,E1 13348.357,E2 13348.357} C_VEL
LIN {X 0,Y 391.882,Z 733.874,A -85,B 0,C 180,E1 13348.106,E2 13348.106} C_VEL
LIN {X 0,Y 387.448,Z 897.622,A -85,B 0,C 180,E1 13344.57,E2 13344.57} C_VEL
LIN {X 0,Y 386.919,Z 915.49,A -85,B 0,C 180,E1 13343.914,E2 13343.914} C_VEL
LIN {X 0,Y 386.053,Z 933.756,A -85,B 0,C 180,E1 13342.942,E2 13342.942} C_VEL
LIN {X 0,Y 385.053,Z 949.93,A -85,B 0,C 180,E1 13341.798,E2 13341.798} C_VEL
LIN {X 0,Y 383.911,Z 965.089,A -85,B 0,C 180,E1 13340.426,E2 13340.426} C_VEL
LIN {X 0,Y 382.654,Z 980.021,A -85,B 0,C 180,E1 13338.748,E2 13338.748} C_VEL
LIN {X 0,Y 381.452,Z 993.201,A -85,B 0,C 180,E1 13336.914,E2 13336.914} C_VEL
LIN {X 0,Y 380.361,Z 1004.78,A -85,B 0,C 180,E1 13334.929,E2 13334.929} C_VEL
LIN {X 0,Y 379.45,Z 1014.939,A -85,B 0,C 180,E1 13332.788,E2 13332.788} C_VEL
LIN {X 0,Y 378.724,Z 1023.63,A -85,B 0,C 180,E1 13330.496,E2 13330.496} C_VEL
LIN {X 0,Y 378.2,Z 1030.749,A -85,B 0,C 180,E1 13328.055,E2 13328.055} C_VEL
LIN {X 0,Y 377.906,Z 1036.302,A -85,B 0,C 180,E1 13325.466,E2 13325.466} C_VEL
LIN {X 0,Y 377.81,Z 1039.748,A -85,B 0,C 180,E1 13323.034,E2 13323.034} C_VEL
LIN {X 0,Y 377.846,Z 1041.617,A -85,B 0,C 180,E1 13320.455,E2 13320.455} C_VEL
LIN {X 0,Y 377.996,Z 1041.751,A -85,B 0,C 180,E1 13317.878,E2 13317.878} C_VEL
LIN {X 0,Y 378.265,Z 1040.225,A -85,B 0,C 180,E1 13315.452,E2 13315.452} C_VEL
LIN {X 0,Y 378.688,Z 1036.987,A -85,B 0,C 180,E1 13313.024,E2 13313.024} C_VEL
LIN {X 0,Y 379.324,Z 1031.976,A -85,B 0,C 180,E1 13310.595,E2 13310.595} C_VEL
LIN {X 0,Y 380.138,Z 1025.465,A -85,B 0,C 180,E1 13308.316,E2 13308.316} C_VEL
LIN {X 0,Y 381.13,Z 1017.094,A -85,B 0,C 180,E1 13306.088,E2 13306.088} C_VEL
LIN {X 0,Y 382.24,Z 1007.396,A -85,B 0,C 180,E1 13304.059,E2 13304.059} C_VEL
LIN {X 0,Y 383.398,Z 996.52,A -85,B 0,C 180,E1 13302.235,E2 13302.235} C_VEL
LIN {X 0,Y 384.58,Z 984.217,A -85,B 0,C 180,E1 13300.563,E2 13300.563} C_VEL
LIN {X 0,Y 385.695,Z 970.166,A -85,B 0,C 180,E1 13299.039,E2 13299.039} C_VEL
LIN {X 0,Y 386.647,Z 955.042,A -85,B 0,C 180,E1 13297.738,E2 13297.738} C_VEL
LIN {X 0,Y 387.417,Z 938.968,A -85,B 0,C 180,E1 13296.671,E2 13296.671} C_VEL
LIN {X 0,Y 387.941,Z 921.083,A -85,B 0,C 180,E1 13295.803,E2 13295.803} C_VEL
LIN {X 0,Y 388.135,Z 902.582,A -85,B 0,C 180,E1 13295.21,E2 13295.21} C_VEL
LIN {X 0,Y 389.947,Z 839.703,A -85,B 0,C 180,E1 13293.705,E2 13293.705} C_VEL
LIN {X 0,Y 394.51,Z 747.388,A -85,B 0,C 180,E1 13291.323,E2 13291.323} C_VEL
LIN {X 0,Y 397.141,Z 735.628,A -85,B 0,C 180,E1 13290.588,E2 13290.588} C_VEL
LIN {X 0,Y 398.624,Z 711.146,A -85,B 0,C 180,E1 13288.477,E2 13288.477} C_VEL
LIN {X 0,Y 399.798,Z 708.668,A -85,B 0,C 180,E1 13288.109,E2 13288.109} C_VEL
LIN {X 0,Y 403.092,Z 704.854,A -85,B 0,C 180,E1 13287.54,E2 13287.54} C_VEL
LIN {X 0,Y 407.167,Z 697.813,A -85,B 0,C 180,E1 13286.944,E2 13286.944} C_VEL
LIN {X 0,Y 408.481,Z 695.738,A -85,B 0,C 180,E1 13286.75,E2 13286.75} C_VEL
LIN {X 0,Y 412.385,Z 691.549,A -85,B 0,C 180,E1 13286.128,E2 13286.128} C_VEL
LIN {X 0,Y 416.977,Z 684.15,A -85,B 0,C 180,E1 13285.494,E2 13285.494} C_VEL
LIN {X 0,Y 418.218,Z 682.394,A -85,B 0,C 180,E1 13285.32,E2 13285.32} C_VEL
LIN {X 0,Y 422.701,Z 677.391,A -85,B 0,C 180,E1 13284.667,E2 13284.667} C_VEL
LIN {X 0,Y 427.839,Z 669.622,A -85,B 0,C 180,E1 13284.003,E2 13284.003} C_VEL
LIN {X 0,Y 432.986,Z 663.854,A -85,B 0,C 180,E1 13283.309,E2 13283.309} C_VEL
LIN {X 0,Y 434.858,Z 661.349,A -85,B 0,C 180,E1 13283.074,E2 13283.074} C_VEL
LIN {X 0,Y 425.579,Z 869.407,A -85,B 0,C 180,E1 13279.06,E2 13279.06} C_VEL
LIN {X 0,Y 423.798,Z 899.627,A -85,B 0,C 180,E1 13278.408,E2 13278.408} C_VEL
LIN {X 0,Y 421.565,Z 922.643,A -85,B 0,C 180,E1 13277.705,E2 13277.705} C_VEL
LIN {X 0,Y 418.735,Z 944.482,A -85,B 0,C 180,E1 13276.793,E2 13276.793} C_VEL
LIN {X 0,Y 415.39,Z 966.517,A -85,B 0,C 180,E1 13275.634,E2 13275.634} C_VEL
LIN {X 0,Y 411.886,Z 986.196,A -85,B 0,C 180,E1 13274.357,E2 13274.357} C_VEL
LIN {X 0,Y 407.678,Z 1007.586,A -85,B 0,C 180,E1 13272.692,E2 13272.692} C_VEL
LIN {X 0,Y 403.639,Z 1026.524,A -85,B 0,C 180,E1 13270.93,E2 13270.93} C_VEL
LIN {X 0,Y 399.199,Z 1046.156,A -85,B 0,C 180,E1 13268.768,E2 13268.768} C_VEL
LIN {X 0,Y 395.073,Z 1063.886,A -85,B 0,C 180,E1 13266.495,E2 13266.495} C_VEL
LIN {X 0,Y 391.05,Z 1080.753,A -85,B 0,C 180,E1 13263.939,E2 13263.939} C_VEL
LIN {X 0,Y 387.085,Z 1097.761,A -85,B 0,C 180,E1 13260.933,E2 13260.933} C_VEL
LIN {X 0,Y 383.929,Z 1112.165,A -85,B 0,C 180,E1 13257.955,E2 13257.955} C_VEL
LIN {X 0,Y 381.285,Z 1124.995,A -85,B 0,C 180,E1 13254.808,E2 13254.808} C_VEL
LIN {X 0,Y 379.175,Z 1136.701,A -85,B 0,C 180,E1 13251.436,E2 13251.436} C_VEL
LIN {X 0,Y 377.862,Z 1145.171,A -85,B 0,C 180,E1 13248.514,E2 13248.514} C_VEL
LIN {X 0,Y 376.816,Z 1153.49,A -85,B 0,C 180,E1 13245.019,E2 13245.019} C_VEL
LIN {X 0,Y 376.298,Z 1159.23,A -85,B 0,C 180,E1 13241.962,E2 13241.962} C_VEL
LIN {X 0,Y 376.018,Z 1164.235,A -85,B 0,C 180,E1 13238.41,E2 13238.41} C_VEL
LIN {X 0,Y 375.923,Z 1166.997,A -85,B 0,C 180,E1 13235.495,E2 13235.495} C_VEL
LIN {X 0,Y 375.922,Z 1168.782,A -85,B 0,C 180,E1 13232.287,E2 13232.287} C_VEL
LIN {X 0,Y 375.904,Z 1169.008,A -85,B 0,C 180,E1 13229.086,E2 13229.086} C_VEL
LIN {X 0,Y 375.911,Z 1168.15,A -85,B 0,C 180,E1 13226.34,E2 13226.34} C_VEL
LIN {X 0,Y 375.944,Z 1165.731,A -85,B 0,C 180,E1 13222.973,E2 13222.973} C_VEL
LIN {X 0,Y 376.097,Z 1162.058,A -85,B 0,C 180,E1 13219.894,E2 13219.894} C_VEL
LIN {X 0,Y 376.465,Z 1157.111,A -85,B 0,C 180,E1 13216.797,E2 13216.797} C_VEL
LIN {X 0,Y 377.243,Z 1149.885,A -85,B 0,C 180,E1 13213.367,E2 13213.367} C_VEL
LIN {X 0,Y 378.443,Z 1141.336,A -85,B 0,C 180,E1 13210.073,E2 13210.073} C_VEL
LIN {X 0,Y 380.114,Z 1131.279,A -85,B 0,C 180,E1 13206.925,E2 13206.925} C_VEL
LIN {X 0,Y 382.517,Z 1118.827,A -85,B 0,C 180,E1 13203.617,E2 13203.617} C_VEL
LIN {X 0,Y 385.288,Z 1105.832,A -85,B 0,C 180,E1 13200.685,E2 13200.685} C_VEL
LIN {X 0,Y 388.639,Z 1091.054,A -85,B 0,C 180,E1 13197.822,E2 13197.822} C_VEL
LIN {X 0,Y 392.477,Z 1074.854,A -85,B 0,C 180,E1 13195.115,E2 13195.115} C_VEL
LIN {X 0,Y 396.525,Z 1057.584,A -85,B 0,C 180,E1 13192.668,E2 13192.668} C_VEL
LIN {X 0,Y 400.752,Z 1039.358,A -85,B 0,C 180,E1 13190.438,E2 13190.438} C_VEL
LIN {X 0,Y 404.965,Z 1020.42,A -85,B 0,C 180,E1 13188.476,E2 13188.476} C_VEL
LIN {X 0,Y 409.298,Z 999.551,A -85,B 0,C 180,E1 13186.65,E2 13186.65} C_VEL
LIN {X 0,Y 413.181,Z 979.17,A -85,B 0,C 180,E1 13185.156,E2 13185.156} C_VEL
LIN {X 0,Y 416.807,Z 957.226,A -85,B 0,C 180,E1 13183.848,E2 13183.848} C_VEL
LIN {X 0,Y 420.091,Z 934.31,A -85,B 0,C 180,E1 13182.755,E2 13182.755} C_VEL
LIN {X 0,Y 422.56,Z 912.748,A -85,B 0,C 180,E1 13181.969,E2 13181.969} C_VEL
LIN {X 0,Y 424.618,Z 888.209,A -85,B 0,C 180,E1 13181.325,E2 13181.325} C_VEL
LIN {X 0,Y 433.45,Z 691.416,A -85,B 0,C 180,E1 13177.507,E2 13177.507} C_VEL
LIN {X 0,Y 436.635,Z 619.616,A -85,B 0,C 180,E1 13176.112,E2 13176.112} C_VEL
LIN {X 0,Y 425.411,Z 602.366,A -85,B 0,C 180,E1 13173.688,E2 13173.688} C_VEL
LIN {X 0,Y 415.629,Z 588.667,A -85,B 0,C 180,E1 13171.387,E2 13171.387} C_VEL
LIN {X 0,Y 407.765,Z 578.269,A -85,B 0,C 180,E1 13169.367,E2 13169.367} C_VEL
LIN {X 0,Y 403.416,Z 572.789,A -85,B 0,C 180,E1 13168.173,E2 13168.173} C_VEL
LIN {X 0,Y 399.657,Z 568.038,A -85,B 0,C 180,E1 13167.085,E2 13167.085} C_VEL
LIN {X 0,Y 395.166,Z 562.609,A -85,B 0,C 180,E1 13165.717,E2 13165.717} C_VEL
LIN {X 0,Y 390.662,Z 557.341,A -85,B 0,C 180,E1 13164.254,E2 13164.254} C_VEL
LIN {X 0,Y 388.561,Z 554.22,A -85,B 0,C 180,E1 13163.185,E2 13163.185} C_VEL
LIN {X 0,Y 387.747,Z 552.506,A -85,B 0,C 180,E1 13162.595,E2 13162.595} C_VEL
LIN {X 0,Y 385.252,Z 548.76,A -85,B 0,C 180,E1 13160.986,E2 13160.986} C_VEL
LIN {X 0,Y 384.523,Z 547.189,A -85,B 0,C 180,E1 13160.391,E2 13160.391} C_VEL
LIN {X 0,Y 381.954,Z 543.761,A -85,B 0,C 180,E1 13158.624,E2 13158.624} C_VEL
LIN {X 0,Y 380.991,Z 541.596,A -85,B 0,C 180,E1 13157.702,E2 13157.702} C_VEL
LIN {X 0,Y 378.227,Z 538.022,A -85,B 0,C 180,E1 13155.485,E2 13155.485} C_VEL
LIN {X 0,Y 377.71,Z 536.221,A -85,B 0,C 180,E1 13154.486,E2 13154.486} C_VEL
LIN {X 0,Y 377.673,Z 535.949,A -85,B 0,C 180,E1 13150.525,E2 13150.525} C_VEL
LIN {X 0,Y 377.68,Z 535.959,A -85,B 0,C 180,E1 13146.383,E2 13146.383} C_VEL
LIN {X 0,Y 377.679,Z 535.992,A -85,B 0,C 180,E1 13142.275,E2 13142.275} C_VEL
LIN {X 0,Y 377.68,Z 536.002,A -85,B 0,C 180,E1 13138.179,E2 13138.179} C_VEL
LIN {X 0,Y 377.681,Z 535.999,A -85,B 0,C 180,E1 13134.073,E2 13134.073} C_VEL
LIN {X 0,Y 377.677,Z 535.973,A -85,B 0,C 180,E1 13129.937,E2 13129.937} C_VEL
LIN {X 0,Y 377.675,Z 535.942,A -85,B 0,C 180,E1 13125.903,E2 13125.903} C_VEL
LIN {X 0,Y 377.725,Z 536.327,A -85,B 0,C 180,E1 13122.913,E2 13122.913} C_VEL
LIN {X 0,Y 379.611,Z 540.243,A -85,B 0,C 180,E1 13120.777,E2 13120.777} C_VEL
LIN {X 0,Y 381.416,Z 542.385,A -85,B 0,C 180,E1 13119.434,E2 13119.434} C_VEL
LIN {X 0,Y 383.364,Z 546.07,A -85,B 0,C 180,E1 13117.779,E2 13117.779} C_VEL
LIN {X 0,Y 384.749,Z 547.696,A -85,B 0,C 180,E1 13116.895,E2 13116.895} C_VEL
LIN {X 0,Y 386.996,Z 551.765,A -85,B 0,C 180,E1 13115.257,E2 13115.257} C_VEL
LIN {X 0,Y 388.146,Z 553.557,A -85,B 0,C 180,E1 13114.52,E2 13114.52} C_VEL
LIN {X 0,Y 391.164,Z 558.779,A -85,B 0,C 180,E1 13112.606,E2 13112.606} C_VEL
LIN {X 0,Y 394.121,Z 564.047,A -85,B 0,C 180,E1 13110.85,E2 13110.85} C_VEL
LIN {X 0,Y 396.725,Z 568.734,A -85,B 0,C 180,E1 13109.396,E2 13109.396} C_VEL
LIN {X 0,Y 401.655,Z 577.876,A -85,B 0,C 180,E1 13106.836,E2 13106.836} C_VEL
LIN {X 0,Y 410.849,Z 590.761,A -85,B 0,C 180,E1 13104.305,E2 13104.305} C_VEL
LIN {X 0,Y 420.406,Z 604.99,A -85,B 0,C 180,E1 13101.952,E2 13101.952} C_VEL
LIN {X 0,Y 430.27,Z 620.664,A -85,B 0,C 180,E1 13099.736,E2 13099.736} C_VEL
LIN {X 0,Y 431.678,Z 623.426,A -85,B 0,C 180,E1 13099.423,E2 13099.423} C_VEL
LIN {X 0,Y 432.989,Z 635.467,A -85,B 0,C 180,E1 13098.897,E2 13098.897} C_VEL
LIN {X 0,Y 424.261,Z 868.168,A -85,B 0,C 180,E1 13094.719,E2 13094.719} C_VEL
LIN {X 0,Y 422.799,Z 900.555,A -85,B 0,C 180,E1 13094.096,E2 13094.096} C_VEL
LIN {X 0,Y 420.884,Z 921.786,A -85,B 0,C 180,E1 13093.493,E2 13093.493} C_VEL
LIN {X 0,Y 418.316,Z 942.803,A -85,B 0,C 180,E1 13092.658,E2 13092.658} C_VEL
LIN {X 0,Y 415.321,Z 962.804,A -85,B 0,C 180,E1 13091.641,E2 13091.641} C_VEL
LIN {X 0,Y 411.818,Z 981.978,A -85,B 0,C 180,E1 13090.41,E2 13090.41} C_VEL
LIN {X 0,Y 407.557,Z 1002.536,A -85,B 0,C 180,E1 13088.796,E2 13088.796} C_VEL
LIN {X 0,Y 403.376,Z 1020.994,A -85,B 0,C 180,E1 13087.037,E2 13087.037} C_VEL
LIN {X 0,Y 399.158,Z 1037.878,A -85,B 0,C 180,E1 13085.1,E2 13085.1} C_VEL
LIN {X 0,Y 394.771,Z 1054.673,A -85,B 0,C 180,E1 13082.821,E2 13082.821} C_VEL
LIN {X 0,Y 392.203,Z 1064.271,A -85,B 0,C 180,E1 13081.32,E2 13081.32} C_VEL
LIN {X 0,Y 389.963,Z 1069.5,A -85,B 0,C 180,E1 13080.531,E2 13080.531} C_VEL
LIN {X 0,Y 381.243,Z 1082.237,A -85,B 0,C 180,E1 13078.624,E2 13078.624} C_VEL
LIN {X 0,Y 379.084,Z 1086.769,A -85,B 0,C 180,E1 13077.732,E2 13077.732} C_VEL
LIN {X 0,Y 375.809,Z 1098.719,A -85,B 0,C 180,E1 13074.858,E2 13074.858} C_VEL
LIN {X 0,Y 373.032,Z 1109.696,A -85,B 0,C 180,E1 13071.709,E2 13071.709} C_VEL
LIN {X 0,Y 370.99,Z 1118.872,A -85,B 0,C 180,E1 13068.543,E2 13068.543} C_VEL
LIN {X 0,Y 369.522,Z 1126.564,A -85,B 0,C 180,E1 13065.216,E2 13065.216} C_VEL
LIN {X 0,Y 368.611,Z 1132.941,A -85,B 0,C 180,E1 13061.701,E2 13061.701} C_VEL
LIN {X 0,Y 368.165,Z 1137.552,A -85,B 0,C 180,E1 13058.276,E2 13058.276} C_VEL
LIN {X 0,Y 367.974,Z 1140.37,A -85,B 0,C 180,E1 13054.988,E2 13054.988} C_VEL
LIN {X 0,Y 367.937,Z 1141.876,A -85,B 0,C 180,E1 13051.557,E2 13051.557} C_VEL
LIN {X 0,Y 367.943,Z 1141.909,A -85,B 0,C 180,E1 13048.599,E2 13048.599} C_VEL
LIN {X 0,Y 367.976,Z 1140.541,A -85,B 0,C 180,E1 13045.168,E2 13045.168} C_VEL
LIN {X 0,Y 368.116,Z 1137.942,A -85,B 0,C 180,E1 13042.038,E2 13042.038} C_VEL
LIN {X 0,Y 368.545,Z 1133.506,A -85,B 0,C 180,E1 13038.577,E2 13038.577} C_VEL
LIN {X 0,Y 369.351,Z 1127.767,A -85,B 0,C 180,E1 13035.258,E2 13035.258} C_VEL
LIN {X 0,Y 370.694,Z 1120.254,A -85,B 0,C 180,E1 13031.929,E2 13031.929} C_VEL
LIN {X 0,Y 372.77,Z 1110.791,A -85,B 0,C 180,E1 13028.551,E2 13028.551} C_VEL
LIN {X 0,Y 375.427,Z 1100.277,A -85,B 0,C 180,E1 13025.451,E2 13025.451} C_VEL
LIN {X 0,Y 378.702,Z 1088.109,A -85,B 0,C 180,E1 13022.481,E2 13022.481} C_VEL
LIN {X 0,Y 382.494,Z 1074.529,A -85,B 0,C 180,E1 13019.701,E2 13019.701} C_VEL
LIN {X 0,Y 386.621,Z 1060.08,A -85,B 0,C 180,E1 13017.193,E2 13017.193} C_VEL
LIN {X 0,Y 391.002,Z 1044.164,A -85,B 0,C 180,E1 13014.875,E2 13014.875} C_VEL
LIN {X 0,Y 395.563,Z 1026.977,A -85,B 0,C 180,E1 13012.771,E2 13012.771} C_VEL
LIN {X 0,Y 399.95,Z 1009.367,A -85,B 0,C 180,E1 13010.95,E2 13010.95} C_VEL
LIN {X 0,Y 404.22,Z 990.225,A -85,B 0,C 180,E1 13009.324,E2 13009.324} C_VEL
LIN {X 0,Y 408.238,Z 969.954,A -85,B 0,C 180,E1 13007.912,E2 13007.912} C_VEL
LIN {X 0,Y 411.776,Z 949.319,A -85,B 0,C 180,E1 13006.757,E2 13006.757} C_VEL
LIN {X 0,Y 414.502,Z 929.18,A -85,B 0,C 180,E1 13005.887,E2 13005.887} C_VEL
LIN {X 0,Y 416.825,Z 907.022,A -85,B 0,C 180,E1 13005.175,E2 13005.175} C_VEL
LIN {X 0,Y 418.29,Z 884.641,A -85,B 0,C 180,E1 13004.679,E2 13004.679} C_VEL
LIN {X 0,Y 427.056,Z 659.536,A -85,B 0,C 180,E1 13000.609,E2 13000.609} C_VEL
LIN {X 0,Y 427.667,Z 641.657,A -85,B 0,C 180,E1 13000.252,E2 13000.252} C_VEL
LIN {X 0,Y 425.946,Z 631.317,A -85,B 0,C 180,E1 12999.679,E2 12999.679} C_VEL
LIN {X 0,Y 420.874,Z 637.631,A -85,B 0,C 180,E1 12998.93,E2 12998.93} C_VEL
LIN {X 0,Y 417.07,Z 641.311,A -85,B 0,C 180,E1 12998.317,E2 12998.317} C_VEL
LIN {X 0,Y 412.191,Z 648.539,A -85,B 0,C 180,E1 12997.573,E2 12997.573} C_VEL
LIN {X 0,Y 407.861,Z 652.947,A -85,B 0,C 180,E1 12996.826,E2 12996.826} C_VEL
LIN {X 0,Y 406.762,Z 654.161,A -85,B 0,C 180,E1 12996.634,E2 12996.634} C_VEL
LIN {X 0,Y 402.14,Z 661.821,A -85,B 0,C 180,E1 12995.885,E2 12995.885} C_VEL
LIN {X 0,Y 398.465,Z 666.008,A -85,B 0,C 180,E1 12995.205,E2 12995.205} C_VEL
LIN {X 0,Y 396.556,Z 667.688,A -85,B 0,C 180,E1 12994.826,E2 12994.826} C_VEL
LIN {X 0,Y 391.723,Z 676.582,A -85,B 0,C 180,E1 12993.986,E2 12993.986} C_VEL
LIN {X 0,Y 388.621,Z 680.489,A -85,B 0,C 180,E1 12993.364,E2 12993.364} C_VEL
LIN {X 0,Y 386.939,Z 682.43,A -85,B 0,C 180,E1 12992.88,E2 12992.88} C_VEL
LIN {X 0,Y 386.319,Z 686.703,A -85,B 0,C 180,E1 12992.395,E2 12992.395} C_VEL
LIN {X 0,Y 384.007,Z 726.479,A -85,B 0,C 180,E1 12988.839,E2 12988.839} C_VEL
LIN {X 0,Y 384.606,Z 734.736,A -85,B 0,C 180,E1 12988.588,E2 12988.588} C_VEL
LIN {X 0,Y 379.926,Z 897.876,A -85,B 0,C 180,E1 12984.975,E2 12984.975} C_VEL
LIN {X 0,Y 379.389,Z 915.934,A -85,B 0,C 180,E1 12984.312,E2 12984.312} C_VEL
LIN {X 0,Y 378.509,Z 934.006,A -85,B 0,C 180,E1 12983.343,E2 12983.343} C_VEL
LIN {X 0,Y 377.472,Z 950.423,A -85,B 0,C 180,E1 12982.177,E2 12982.177} C_VEL
LIN {X 0,Y 376.286,Z 965.779,A -85,B 0,C 180,E1 12980.777,E2 12980.777} C_VEL
LIN {X 0,Y 375.002,Z 980.556,A -85,B 0,C 180,E1 12979.101,E2 12979.101} C_VEL
LIN {X 0,Y 373.765,Z 993.825,A -85,B 0,C 180,E1 12977.251,E2 12977.251} C_VEL
LIN {X 0,Y 372.63,Z 1005.447,A -85,B 0,C 180,E1 12975.246,E2 12975.246} C_VEL
LIN {X 0,Y 371.665,Z 1015.759,A -85,B 0,C 180,E1 12973.061,E2 12973.061} C_VEL
LIN {X 0,Y 370.904,Z 1024.631,A -85,B 0,C 180,E1 12970.72,E2 12970.72} C_VEL
LIN {X 0,Y 370.346,Z 1031.872,A -85,B 0,C 180,E1 12968.227,E2 12968.227} C_VEL
LIN {X 0,Y 370.045,Z 1037.255,A -85,B 0,C 180,E1 12965.738,E2 12965.738} C_VEL
LIN {X 0,Y 369.938,Z 1040.933,A -85,B 0,C 180,E1 12963.254,E2 12963.254} C_VEL
LIN {X 0,Y 369.973,Z 1042.997,A -85,B 0,C 180,E1 12960.635,E2 12960.635} C_VEL
LIN {X 0,Y 370.129,Z 1043.296,A -85,B 0,C 180,E1 12957.988,E2 12957.988} C_VEL
LIN {X 0,Y 370.445,Z 1041.807,A -85,B 0,C 180,E1 12955.356,E2 12955.356} C_VEL
LIN {X 0,Y 370.912,Z 1038.626,A -85,B 0,C 180,E1 12952.877,E2 12952.877} C_VEL
LIN {X 0,Y 371.601,Z 1033.635,A -85,B 0,C 180,E1 12950.397,E2 12950.397} C_VEL
LIN {X 0,Y 372.482,Z 1027.162,A -85,B 0,C 180,E1 12948.072,E2 12948.072} C_VEL
LIN {X 0,Y 373.502,Z 1019.255,A -85,B 0,C 180,E1 12945.901,E2 12945.901} C_VEL
LIN {X 0,Y 374.634,Z 1009.909,A -85,B 0,C 180,E1 12943.886,E2 12943.886} C_VEL
LIN {X 0,Y 375.97,Z 998.259,A -85,B 0,C 180,E1 12941.872,E2 12941.872} C_VEL
LIN {X 0,Y 377.217,Z 985.921,A -85,B 0,C 180,E1 12940.168,E2 12940.168} C_VEL
LIN {X 0,Y 378.398,Z 971.868,A -85,B 0,C 180,E1 12938.615,E2 12938.615} C_VEL
LIN {X 0,Y 379.438,Z 956.442,A -85,B 0,C 180,E1 12937.264,E2 12937.264} C_VEL
LIN {X 0,Y 380.253,Z 939.765,A -85,B 0,C 180,E1 12936.152,E2 12936.152} C_VEL
LIN {X 0,Y 380.807,Z 922.201,A -85,B 0,C 180,E1 12935.288,E2 12935.288} C_VEL
LIN {X 0,Y 381.012,Z 902.859,A -85,B 0,C 180,E1 12934.668,E2 12934.668} C_VEL
LIN {X 0,Y 383.089,Z 840.711,A -85,B 0,C 180,E1 12933.106,E2 12933.106} C_VEL
LIN {X 0,Y 388.07,Z 750.26,A -85,B 0,C 180,E1 12930.67,E2 12930.67} C_VEL
LIN {X 0,Y 391.032,Z 736.877,A -85,B 0,C 180,E1 12929.839,E2 12929.839} C_VEL
LIN {X 0,Y 391.76,Z 730.502,A -85,B 0,C 180,E1 12929.222,E2 12929.222} C_VEL
LIN {X 0,Y 395.319,Z 725.92,A -85,B 0,C 180,E1 12928.483,E2 12928.483} C_VEL
LIN {X 0,Y 399.605,Z 718.6,A -85,B 0,C 180,E1 12927.817,E2 12927.817} C_VEL
LIN {X 0,Y 401.447,Z 715.422,A -85,B 0,C 180,E1 12927.539,E2 12927.539} C_VEL
LIN {X 0,Y 405.386,Z 710.999,A -85,B 0,C 180,E1 12926.886,E2 12926.886} C_VEL
LIN {X 0,Y 409.92,Z 703.575,A -85,B 0,C 180,E1 12926.233,E2 12926.233} C_VEL
LIN {X 0,Y 411.074,Z 701.781,A -85,B 0,C 180,E1 12926.068,E2 12926.068} C_VEL
LIN {X 0,Y 415.497,Z 696.743,A -85,B 0,C 180,E1 12925.396,E2 12925.396} C_VEL
LIN {X 0,Y 420.939,Z 688.372,A -85,B 0,C 180,E1 12924.663,E2 12924.663} C_VEL
LIN {X 0,Y 426.04,Z 682.445,A -85,B 0,C 180,E1 12923.952,E2 12923.952} C_VEL
LIN {X 0,Y 428.986,Z 678.192,A -85,B 0,C 180,E1 12923.576,E2 12923.576} C_VEL
LIN {X 0,Y 419.562,Z 881.217,A -85,B 0,C 180,E1 12919.623,E2 12919.623} C_VEL
LIN {X 0,Y 417.894,Z 904.016,A -85,B 0,C 180,E1 12919.08,E2 12919.08} C_VEL
LIN {X 0,Y 415.323,Z 927.485,A -85,B 0,C 180,E1 12918.304,E2 12918.304} C_VEL
LIN {X 0,Y 412.518,Z 947.951,A -85,B 0,C 180,E1 12917.411,E2 12917.411} C_VEL
LIN {X 0,Y 408.822,Z 970.307,A -85,B 0,C 180,E1 12916.177,E2 12916.177} C_VEL
LIN {X 0,Y 405.034,Z 990.582,A -85,B 0,C 180,E1 12914.812,E2 12914.812} C_VEL
LIN {X 0,Y 400.7,Z 1011.052,A -85,B 0,C 180,E1 12913.134,E2 12913.134} C_VEL
LIN {X 0,Y 396.216,Z 1030.982,A -85,B 0,C 180,E1 12911.196,E2 12911.196} C_VEL
LIN {X 0,Y 391.928,Z 1048.804,A -85,B 0,C 180,E1 12909.147,E2 12909.147} C_VEL
LIN {X 0,Y 387.251,Z 1067.587,A -85,B 0,C 180,E1 12906.615,E2 12906.615} C_VEL
LIN {X 0,Y 383.094,Z 1084.438,A -85,B 0,C 180,E1 12903.954,E2 12903.954} C_VEL
LIN {X 0,Y 379.302,Z 1099.698,A -85,B 0,C 180,E1 12901.109,E2 12901.109} C_VEL
LIN {X 0,Y 375.885,Z 1114.376,A -85,B 0,C 180,E1 12897.915,E2 12897.915} C_VEL
LIN {X 0,Y 373.329,Z 1126.317,A -85,B 0,C 180,E1 12894.865,E2 12894.865} C_VEL
LIN {X 0,Y 371.196,Z 1137.458,A -85,B 0,C 180,E1 12891.49,E2 12891.49} C_VEL
LIN {X 0,Y 369.71,Z 1146.831,A -85,B 0,C 180,E1 12888.12,E2 12888.12} C_VEL
LIN {X 0,Y 368.755,Z 1154.25,A -85,B 0,C 180,E1 12884.766,E2 12884.766} C_VEL
LIN {X 0,Y 368.236,Z 1160.208,A -85,B 0,C 180,E1 12881.42,E2 12881.42} C_VEL
LIN {X 0,Y 368.01,Z 1164.407,A -85,B 0,C 180,E1 12878.122,E2 12878.122} C_VEL
LIN {X 0,Y 367.929,Z 1167.162,A -85,B 0,C 180,E1 12874.989,E2 12874.989} C_VEL
LIN {X 0,Y 367.926,Z 1168.622,A -85,B 0,C 180,E1 12871.557,E2 12871.557} C_VEL
LIN {X 0,Y 367.925,Z 1168.647,A -85,B 0,C 180,E1 12868.599,E2 12868.599} C_VEL
LIN {X 0,Y 367.927,Z 1167.282,A -85,B 0,C 180,E1 12865.167,E2 12865.167} C_VEL
LIN {X 0,Y 368.009,Z 1164.417,A -85,B 0,C 180,E1 12861.878,E2 12861.878} C_VEL
LIN {X 0,Y 368.237,Z 1160.191,A -85,B 0,C 180,E1 12858.567,E2 12858.567} C_VEL
LIN {X 0,Y 368.754,Z 1154.263,A -85,B 0,C 180,E1 12855.234,E2 12855.234} C_VEL
LIN {X 0,Y 369.71,Z 1146.831,A -85,B 0,C 180,E1 12851.88,E2 12851.88} C_VEL
LIN {X 0,Y 371.196,Z 1137.463,A -85,B 0,C 180,E1 12848.51,E2 12848.51} C_VEL
LIN {X 0,Y 373.331,Z 1126.322,A -85,B 0,C 180,E1 12845.135,E2 12845.135} C_VEL
LIN {X 0,Y 375.885,Z 1114.376,A -85,B 0,C 180,E1 12842.085,E2 12842.085} C_VEL
LIN {X 0,Y 379.299,Z 1099.692,A -85,B 0,C 180,E1 12838.891,E2 12838.891} C_VEL
LIN {X 0,Y 383.094,Z 1084.428,A -85,B 0,C 180,E1 12836.046,E2 12836.046} C_VEL
LIN {X 0,Y 387.25,Z 1067.571,A -85,B 0,C 180,E1 12833.385,E2 12833.385} C_VEL
LIN {X 0,Y 391.918,Z 1048.795,A -85,B 0,C 180,E1 12830.855,E2 12830.855} C_VEL
LIN {X 0,Y 396.21,Z 1030.943,A -85,B 0,C 180,E1 12828.803,E2 12828.803} C_VEL
LIN {X 0,Y 400.694,Z 1011.001,A -85,B 0,C 180,E1 12826.865,E2 12826.865} C_VEL
LIN {X 0,Y 405.027,Z 990.523,A -85,B 0,C 180,E1 12825.187,E2 12825.187} C_VEL
LIN {X 0,Y 408.814,Z 970.232,A -85,B 0,C 180,E1 12823.822,E2 12823.822} C_VEL
LIN {X 0,Y 412.509,Z 947.842,A -85,B 0,C 180,E1 12822.587,E2 12822.587} C_VEL
LIN {X 0,Y 415.319,Z 927.301,A -85,B 0,C 180,E1 12821.692,E2 12821.692} C_VEL
LIN {X 0,Y 417.895,Z 903.646,A -85,B 0,C 180,E1 12820.914,E2 12820.914} C_VEL
LIN {X 0,Y 419.577,Z 880.491,A -85,B 0,C 180,E1 12820.366,E2 12820.366} C_VEL
LIN {X 0,Y 429.322,Z 670.802,A -85,B 0,C 180,E1 12816.287,E2 12816.287} C_VEL
LIN {X 0,Y 431.429,Z 623.46,A -85,B 0,C 180,E1 12815.346,E2 12815.346} C_VEL
LIN {X 0,Y 420.68,Z 606.877,A -85,B 0,C 180,E1 12812.934,E2 12812.934} C_VEL
LIN {X 0,Y 409.692,Z 591.346,A -85,B 0,C 180,E1 12810.222,E2 12810.222} C_VEL
LIN {X 0,Y 400.955,Z 580.044,A -85,B 0,C 180,E1 12807.836,E2 12807.836} C_VEL
LIN {X 0,Y 396.699,Z 574.676,A -85,B 0,C 180,E1 12806.575,E2 12806.575} C_VEL
LIN {X 0,Y 392.5,Z 569.519,A -85,B 0,C 180,E1 12805.257,E2 12805.257} C_VEL
LIN {X 0,Y 388.174,Z 564.379,A -85,B 0,C 180,E1 12803.813,E2 12803.813} C_VEL
LIN {X 0,Y 383.503,Z 558.926,A -85,B 0,C 180,E1 12802.131,E2 12802.131} C_VEL
LIN {X 0,Y 381.465,Z 556.512,A -85,B 0,C 180,E1 12801.205,E2 12801.205} C_VEL
LIN {X 0,Y 380.057,Z 553.673,A -85,B 0,C 180,E1 12800.082,E2 12800.082} C_VEL
LIN {X 0,Y 377.688,Z 550.302,A -85,B 0,C 180,E1 12798.362,E2 12798.362} C_VEL
LIN {X 0,Y 376.723,Z 548.28,A -85,B 0,C 180,E1 12797.452,E2 12797.452} C_VEL
LIN {X 0,Y 374.054,Z 544.57,A -85,B 0,C 180,E1 12795.186,E2 12795.186} C_VEL
LIN {X 0,Y 373.117,Z 542.637,A -85,B 0,C 180,E1 12794.114,E2 12794.114} C_VEL
LIN {X 0,Y 370.238,Z 538.916,A -85,B 0,C 180,E1 12791.054,E2 12791.054} C_VEL
LIN {X 0,Y 369.768,Z 537.166,A -85,B 0,C 180,E1 12789.651,E2 12789.651} C_VEL
LIN {X 0,Y 369.734,Z 536.962,A -85,B 0,C 180,E1 12785.898,E2 12785.898} C_VEL
LIN {X 0,Y 369.736,Z 536.991,A -85,B 0,C 180,E1 12781.704,E2 12781.704} C_VEL
LIN {X 0,Y 369.735,Z 536.986,A -85,B 0,C 180,E1 12777.52,E2 12777.52} C_VEL
LIN {X 0,Y 369.734,Z 536.977,A -85,B 0,C 180,E1 12773.322,E2 12773.322} C_VEL
LIN {X 0,Y 369.731,Z 536.944,A -85,B 0,C 180,E1 12769.245,E2 12769.245} C_VEL
LIN {X 0,Y 369.811,Z 537.411,A -85,B 0,C 180,E1 12767.508,E2 12767.508} C_VEL
LIN {X 0,Y 372.117,Z 541.744,A -85,B 0,C 180,E1 12764.253,E2 12764.253} C_VEL
LIN {X 0,Y 373.597,Z 543.455,A -85,B 0,C 180,E1 12762.878,E2 12762.878} C_VEL
LIN {X 0,Y 375.727,Z 547.308,A -85,B 0,C 180,E1 12760.732,E2 12760.732} C_VEL
LIN {X 0,Y 377.124,Z 548.956,A -85,B 0,C 180,E1 12759.676,E2 12759.676} C_VEL
LIN {X 0,Y 379.019,Z 552.654,A -85,B 0,C 180,E1 12758,E2 12758} C_VEL
LIN {X 0,Y 380.376,Z 554.29,A -85,B 0,C 180,E1 12757.105,E2 12757.105} C_VEL
LIN {X 0,Y 382.661,Z 558.412,A -85,B 0,C 180,E1 12755.408,E2 12755.408} C_VEL
LIN {X 0,Y 383.71,Z 560.165,A -85,B 0,C 180,E1 12754.7,E2 12754.7} C_VEL
LIN {X 0,Y 386.683,Z 565.404,A -85,B 0,C 180,E1 12752.762,E2 12752.762} C_VEL
LIN {X 0,Y 389.604,Z 570.684,A -85,B 0,C 180,E1 12750.985,E2 12750.985} C_VEL
LIN {X 0,Y 392.169,Z 575.409,A -85,B 0,C 180,E1 12749.511,E2 12749.511} C_VEL
LIN {X 0,Y 394.536,Z 578.926,A -85,B 0,C 180,E1 12748.572,E2 12748.572} C_VEL
LIN {X 0,Y 404.781,Z 593.03,A -85,B 0,C 180,E1 12745.576,E2 12745.576} C_VEL
LIN {X 0,Y 414.76,Z 607.841,A -85,B 0,C 180,E1 12742.981,E2 12742.981} C_VEL
LIN {X 0,Y 425.489,Z 624.876,A -85,B 0,C 180,E1 12740.466,E2 12740.466} C_VEL
LIN {X 0,Y 427.052,Z 627.985,A -85,B 0,C 180,E1 12740.106,E2 12740.106} C_VEL
LIN {X 0,Y 427.971,Z 637.078,A -85,B 0,C 180,E1 12739.708,E2 12739.708} C_VEL
LIN {X 0,Y 418.792,Z 869.745,A -85,B 0,C 180,E1 12735.495,E2 12735.495} C_VEL
LIN {X 0,Y 417.293,Z 900.854,A -85,B 0,C 180,E1 12734.888,E2 12734.888} C_VEL
LIN {X 0,Y 415.278,Z 922.283,A -85,B 0,C 180,E1 12734.273,E2 12734.273} C_VEL
LIN {X 0,Y 412.618,Z 943.066,A -85,B 0,C 180,E1 12733.44,E2 12733.44} C_VEL
LIN {X 0,Y 409.398,Z 963.58,A -85,B 0,C 180,E1 12732.382,E2 12732.382} C_VEL
LIN {X 0,Y 405.763,Z 982.68,A -85,B 0,C 180,E1 12731.142,E2 12731.142} C_VEL
LIN {X 0,Y 401.556,Z 1002.157,A -85,B 0,C 180,E1 12729.601,E2 12729.601} C_VEL
LIN {X 0,Y 397.299,Z 1020.15,A -85,B 0,C 180,E1 12727.884,E2 12727.884} C_VEL
LIN {X 0,Y 392.853,Z 1037.244,A -85,B 0,C 180,E1 12725.92,E2 12725.92} C_VEL
LIN {X 0,Y 388.244,Z 1054.137,A -85,B 0,C 180,E1 12723.621,E2 12723.621} C_VEL
LIN {X 0,Y 384.054,Z 1069.102,A -85,B 0,C 180,E1 12721.204,E2 12721.204} C_VEL
LIN {X 0,Y 380.107,Z 1082.986,A -85,B 0,C 180,E1 12718.528,E2 12718.528} C_VEL
LIN {X 0,Y 379.084,Z 1086.769,A -85,B 0,C 180,E1 12717.732,E2 12717.732} C_VEL
LIN {X 0,Y 376.955,Z 1091.146,A -85,B 0,C 180,E1 12716.81,E2 12716.81} C_VEL
LIN {X 0,Y 368.515,Z 1101.994,A -85,B 0,C 180,E1 12714.539,E2 12714.539} C_VEL
LIN {X 0,Y 366.582,Z 1105.707,A -85,B 0,C 180,E1 12713.531,E2 12713.531} C_VEL
LIN {X 0,Y 364.04,Z 1115.719,A -85,B 0,C 180,E1 12710.247,E2 12710.247} C_VEL
LIN {X 0,Y 362.204,Z 1124.205,A -85,B 0,C 180,E1 12706.849,E2 12706.849} C_VEL
LIN {X 0,Y 361.018,Z 1130.84,A -85,B 0,C 180,E1 12703.453,E2 12703.453} C_VEL
LIN {X 0,Y 360.336,Z 1136.12,A -85,B 0,C 180,E1 12699.906,E2 12699.906} C_VEL
LIN {X 0,Y 360.064,Z 1139.667,A -85,B 0,C 180,E1 12696.537,E2 12696.537} C_VEL
LIN {X 0,Y 359.955,Z 1141.664,A -85,B 0,C 180,E1 12693.185,E2 12693.185} C_VEL
LIN {X 0,Y 359.949,Z 1142.372,A -85,B 0,C 180,E1 12689.841,E2 12689.841} C_VEL
LIN {X 0,Y 359.957,Z 1141.637,A -85,B 0,C 180,E1 12686.656,E2 12686.656} C_VEL
LIN {X 0,Y 360.069,Z 1139.603,A -85,B 0,C 180,E1 12683.302,E2 12683.302} C_VEL
LIN {X 0,Y 360.327,Z 1136.227,A -85,B 0,C 180,E1 12680.091,E2 12680.091} C_VEL
LIN {X 0,Y 361.026,Z 1130.802,A -85,B 0,C 180,E1 12676.433,E2 12676.433} C_VEL
LIN {X 0,Y 362.243,Z 1124.057,A -85,B 0,C 180,E1 12672.987,E2 12672.987} C_VEL
LIN {X 0,Y 364.09,Z 1115.521,A -85,B 0,C 180,E1 12669.588,E2 12669.588} C_VEL
LIN {X 0,Y 366.742,Z 1105.111,A -85,B 0,C 180,E1 12666.203,E2 12666.203} C_VEL
LIN {X 0,Y 369.975,Z 1093.629,A -85,B 0,C 180,E1 12663.104,E2 12663.104} C_VEL
LIN {X 0,Y 373.603,Z 1081.222,A -85,B 0,C 180,E1 12660.323,E2 12660.323} C_VEL
LIN {X 0,Y 378.004,Z 1066.412,A -85,B 0,C 180,E1 12657.523,E2 12657.523} C_VEL
LIN {X 0,Y 382.563,Z 1051.098,A -85,B 0,C 180,E1 12655.084,E2 12655.084} C_VEL
LIN {X 0,Y 387.04,Z 1035.204,A -85,B 0,C 180,E1 12652.964,E2 12652.964} C_VEL
LIN {X 0,Y 392.052,Z 1016.41,A -85,B 0,C 180,E1 12650.861,E2 12650.861} C_VEL
LIN {X 0,Y 396.632,Z 997.863,A -85,B 0,C 180,E1 12649.136,E2 12649.136} C_VEL
LIN {X 0,Y 400.821,Z 978.433,A -85,B 0,C 180,E1 12647.66,E2 12647.66} C_VEL
LIN {X 0,Y 404.78,Z 957.339,A -85,B 0,C 180,E1 12646.365,E2 12646.365} C_VEL
LIN {X 0,Y 408.062,Z 936.396,A -85,B 0,C 180,E1 12645.35,E2 12645.35} C_VEL
LIN {X 0,Y 410.585,Z 915.42,A -85,B 0,C 180,E1 12644.596,E2 12644.596} C_VEL
LIN {X 0,Y 412.513,Z 892.302,A -85,B 0,C 180,E1 12644.012,E2 12644.012} C_VEL
LIN {X 0,Y 421.992,Z 663.291,A -85,B 0,C 180,E1 12639.821,E2 12639.821} C_VEL
LIN {X 0,Y 422.795,Z 644.342,A -85,B 0,C 180,E1 12639.462,E2 12639.462} C_VEL
LIN {X 0,Y 419.426,Z 647.689,A -85,B 0,C 180,E1 12638.936,E2 12638.936} C_VEL
LIN {X 0,Y 414.261,Z 655.011,A -85,B 0,C 180,E1 12638.162,E2 12638.162} C_VEL
LIN {X 0,Y 409.064,Z 660.485,A -85,B 0,C 180,E1 12637.292,E2 12637.292} C_VEL
LIN {X 0,Y 404.166,Z 668.22,A -85,B 0,C 180,E1 12636.511,E2 12636.511} C_VEL
LIN {X 0,Y 399.982,Z 672.878,A -85,B 0,C 180,E1 12635.755,E2 12635.755} C_VEL
LIN {X 0,Y 398.617,Z 674.282,A -85,B 0,C 180,E1 12635.498,E2 12635.498} C_VEL
LIN {X 0,Y 393.756,Z 682.79,A -85,B 0,C 180,E1 12634.667,E2 12634.667} C_VEL
LIN {X 0,Y 390.159,Z 687.229,A -85,B 0,C 180,E1 12633.964,E2 12633.964} C_VEL
LIN {X 0,Y 388.152,Z 689.16,A -85,B 0,C 180,E1 12633.542,E2 12633.542} C_VEL
LIN {X 0,Y 383.356,Z 698.393,A -85,B 0,C 180,E1 12632.654,E2 12632.654} C_VEL
LIN {X 0,Y 380.249,Z 702.684,A -85,B 0,C 180,E1 12631.995,E2 12631.995} C_VEL
LIN {X 0,Y 378.521,Z 704.848,A -85,B 0,C 180,E1 12631.486,E2 12631.486} C_VEL
LIN {X 0,Y 377.847,Z 709.269,A -85,B 0,C 180,E1 12630.977,E2 12630.977} C_VEL
LIN {X 0,Y 376.8,Z 727.628,A -85,B 0,C 180,E1 12629.335,E2 12629.335} C_VEL
LIN {X 0,Y 377.356,Z 735.705,A -85,B 0,C 180,E1 12629.087,E2 12629.087} C_VEL
LIN {X 0,Y 372.394,Z 899.009,A -85,B 0,C 180,E1 12625.366,E2 12625.366} C_VEL
LIN {X 0,Y 371.831,Z 917.14,A -85,B 0,C 180,E1 12624.686,E2 12624.686} C_VEL
LIN {X 0,Y 370.98,Z 934.188,A -85,B 0,C 180,E1 12623.762,E2 12623.762} C_VEL
LIN {X 0,Y 369.902,Z 950.834,A -85,B 0,C 180,E1 12622.572,E2 12622.572} C_VEL
LIN {X 0,Y 368.672,Z 966.431,A -85,B 0,C 180,E1 12621.144,E2 12621.144} C_VEL
LIN {X 0,Y 367.309,Z 981.642,A -85,B 0,C 180,E1 12619.397,E2 12619.397} C_VEL
LIN {X 0,Y 366.013,Z 995.12,A -85,B 0,C 180,E1 12617.488,E2 12617.488} C_VEL
LIN {X 0,Y 364.824,Z 1006.905,A -85,B 0,C 180,E1 12615.418,E2 12615.418} C_VEL
LIN {X 0,Y 363.83,Z 1017.256,A -85,B 0,C 180,E1 12613.185,E2 12613.185} C_VEL
LIN {X 0,Y 363.039,Z 1026.132,A -85,B 0,C 180,E1 12610.795,E2 12610.795} C_VEL
LIN {X 0,Y 362.468,Z 1033.396,A -85,B 0,C 180,E1 12608.247,E2 12608.247} C_VEL
LIN {X 0,Y 362.164,Z 1038.792,A -85,B 0,C 180,E1 12605.704,E2 12605.704} C_VEL
LIN {X 0,Y 362.062,Z 1042.462,A -85,B 0,C 180,E1 12603.167,E2 12603.167} C_VEL
LIN {X 0,Y 362.111,Z 1044.512,A -85,B 0,C 180,E1 12600.475,E2 12600.475} C_VEL
LIN {X 0,Y 362.298,Z 1044.793,A -85,B 0,C 180,E1 12597.786,E2 12597.786} C_VEL
LIN {X 0,Y 362.628,Z 1043.397,A -85,B 0,C 180,E1 12595.256,E2 12595.256} C_VEL
LIN {X 0,Y 363.141,Z 1040.277,A -85,B 0,C 180,E1 12592.724,E2 12592.724} C_VEL
LIN {X 0,Y 363.894,Z 1035.346,A -85,B 0,C 180,E1 12590.192,E2 12590.192} C_VEL
LIN {X 0,Y 364.841,Z 1028.892,A -85,B 0,C 180,E1 12587.818,E2 12587.818} C_VEL
LIN {X 0,Y 365.938,Z 1021.023,A -85,B 0,C 180,E1 12585.603,E2 12585.603} C_VEL
LIN {X 0,Y 367.155,Z 1011.723,A -85,B 0,C 180,E1 12583.548,E2 12583.548} C_VEL
LIN {X 0,Y 368.569,Z 1000.059,A -85,B 0,C 180,E1 12581.495,E2 12581.495} C_VEL
LIN {X 0,Y 369.899,Z 987.769,A -85,B 0,C 180,E1 12579.758,E2 12579.758} C_VEL
LIN {X 0,Y 371.144,Z 973.69,A -85,B 0,C 180,E1 12578.176,E2 12578.176} C_VEL
LIN {X 0,Y 372.233,Z 958.704,A -85,B 0,C 180,E1 12576.827,E2 12576.827} C_VEL
LIN {X 0,Y 373.1,Z 942.338,A -85,B 0,C 180,E1 12575.702,E2 12575.702} C_VEL
LIN {X 0,Y 373.719,Z 924.367,A -85,B 0,C 180,E1 12574.785,E2 12574.785} C_VEL
LIN {X 0,Y 373.976,Z 904.744,A -85,B 0,C 180,E1 12574.127,E2 12574.127} C_VEL
LIN {X 0,Y 376.131,Z 846.312,A -85,B 0,C 180,E1 12572.589,E2 12572.589} C_VEL
LIN {X 0,Y 380.557,Z 772.52,A -85,B 0,C 180,E1 12570.514,E2 12570.514} C_VEL
LIN {X 0,Y 381.94,Z 765.27,A -85,B 0,C 180,E1 12570.173,E2 12570.173} C_VEL
LIN {X 0,Y 385.557,Z 755.242,A -85,B 0,C 180,E1 12569.656,E2 12569.656} C_VEL
LIN {X 0,Y 387.416,Z 750.109,A -85,B 0,C 180,E1 12569.409,E2 12569.409} C_VEL
LIN {X 0,Y 392.745,Z 738.296,A -85,B 0,C 180,E1 12568.627,E2 12568.627} C_VEL
LIN {X 0,Y 394.28,Z 735.75,A -85,B 0,C 180,E1 12568.379,E2 12568.379} C_VEL
LIN {X 0,Y 398.253,Z 731.052,A -85,B 0,C 180,E1 12567.694,E2 12567.694} C_VEL
LIN {X 0,Y 403.015,Z 722.9,A -85,B 0,C 180,E1 12566.985,E2 12566.985} C_VEL
LIN {X 0,Y 404.135,Z 721.278,A -85,B 0,C 180,E1 12566.813,E2 12566.813} C_VEL
LIN {X 0,Y 408.69,Z 715.821,A -85,B 0,C 180,E1 12566.097,E2 12566.097} C_VEL
LIN {X 0,Y 413.901,Z 707.58,A -85,B 0,C 180,E1 12565.369,E2 12565.369} C_VEL
LIN {X 0,Y 418.858,Z 701.668,A -85,B 0,C 180,E1 12564.65,E2 12564.65} C_VEL
LIN {X 0,Y 423.145,Z 695.108,A -85,B 0,C 180,E1 12564.091,E2 12564.091} C_VEL
LIN {X 0,Y 413.749,Z 887.748,A -85,B 0,C 180,E1 12560.295,E2 12560.295} C_VEL
LIN {X 0,Y 411.653,Z 911.697,A -85,B 0,C 180,E1 12559.667,E2 12559.667} C_VEL
LIN {X 0,Y 409.091,Z 932.571,A -85,B 0,C 180,E1 12558.91,E2 12558.91} C_VEL
LIN {X 0,Y 405.538,Z 955.9,A -85,B 0,C 180,E1 12557.807,E2 12557.807} C_VEL
LIN {X 0,Y 401.668,Z 977.552,A -85,B 0,C 180,E1 12556.521,E2 12556.521} C_VEL
LIN {X 0,Y 397.385,Z 998.267,A -85,B 0,C 180,E1 12554.994,E2 12554.994} C_VEL
LIN {X 0,Y 392.833,Z 1018.552,A -85,B 0,C 180,E1 12553.21,E2 12553.21} C_VEL
LIN {X 0,Y 388.425,Z 1036.612,A -85,B 0,C 180,E1 12551.32,E2 12551.32} C_VEL
LIN {X 0,Y 383.449,Z 1056.022,A -85,B 0,C 180,E1 12548.934,E2 12548.934} C_VEL
LIN {X 0,Y 378.908,Z 1073.477,A -85,B 0,C 180,E1 12546.407,E2 12546.407} C_VEL
LIN {X 0,Y 374.707,Z 1089.255,A -85,B 0,C 180,E1 12543.713,E2 12543.713} C_VEL
LIN {X 0,Y 370.96,Z 1103.975,A -85,B 0,C 180,E1 12540.805,E2 12540.805} C_VEL
LIN {X 0,Y 367.687,Z 1117.263,A -85,B 0,C 180,E1 12537.711,E2 12537.711} C_VEL
LIN {X 0,Y 364.882,Z 1129.817,A -85,B 0,C 180,E1 12534.27,E2 12534.27} C_VEL
LIN {X 0,Y 362.925,Z 1139.927,A -85,B 0,C 180,E1 12530.987,E2 12530.987} C_VEL
LIN {X 0,Y 361.501,Z 1148.647,A -85,B 0,C 180,E1 12527.547,E2 12527.547} C_VEL
LIN {X 0,Y 360.654,Z 1155.452,A -85,B 0,C 180,E1 12524.285,E2 12524.285} C_VEL
LIN {X 0,Y 360.183,Z 1160.928,A -85,B 0,C 180,E1 12520.881,E2 12520.881} C_VEL
LIN {X 0,Y 359.985,Z 1164.587,A -85,B 0,C 180,E1 12517.822,E2 12517.822} C_VEL
LIN {X 0,Y 359.932,Z 1167.339,A -85,B 0,C 180,E1 12514.301,E2 12514.301} C_VEL
LIN {X 0,Y 359.928,Z 1168.377,A -85,B 0,C 180,E1 12511.273,E2 12511.273} C_VEL
LIN {X 0,Y 359.931,Z 1168.307,A -85,B 0,C 180,E1 12508.249,E2 12508.249} C_VEL
LIN {X 0,Y 359.931,Z 1166.742,A -85,B 0,C 180,E1 12504.74,E2 12504.74} C_VEL
LIN {X 0,Y 360.022,Z 1163.921,A -85,B 0,C 180,E1 12501.536,E2 12501.536} C_VEL
LIN {X 0,Y 360.303,Z 1159.308,A -85,B 0,C 180,E1 12497.987,E2 12497.987} C_VEL
LIN {X 0,Y 360.866,Z 1153.537,A -85,B 0,C 180,E1 12494.739,E2 12494.739} C_VEL
LIN {X 0,Y 361.985,Z 1145.553,A -85,B 0,C 180,E1 12491.145,E2 12491.145} C_VEL
LIN {X 0,Y 363.548,Z 1136.563,A -85,B 0,C 180,E1 12487.865,E2 12487.865} C_VEL
LIN {X 0,Y 365.993,Z 1124.699,A -85,B 0,C 180,E1 12484.255,E2 12484.255} C_VEL
LIN {X 0,Y 368.853,Z 1112.479,A -85,B 0,C 180,E1 12481.111,E2 12481.111} C_VEL
LIN {X 0,Y 372.32,Z 1098.449,A -85,B 0,C 180,E1 12478.059,E2 12478.059} C_VEL
LIN {X 0,Y 376.369,Z 1083.007,A -85,B 0,C 180,E1 12475.168,E2 12475.168} C_VEL
LIN {X 0,Y 380.679,Z 1066.569,A -85,B 0,C 180,E1 12472.552,E2 12472.552} C_VEL
LIN {X 0,Y 385.463,Z 1048.226,A -85,B 0,C 180,E1 12470.063,E2 12470.063} C_VEL
LIN {X 0,Y 390.079,Z 1029.922,A -85,B 0,C 180,E1 12467.941,E2 12467.941} C_VEL
LIN {X 0,Y 394.668,Z 1010.385,A -85,B 0,C 180,E1 12466.04,E2 12466.04} C_VEL
LIN {X 0,Y 399.141,Z 990.088,A -85,B 0,C 180,E1 12464.37,E2 12464.37} C_VEL
LIN {X 0,Y 403.029,Z 970.104,A -85,B 0,C 180,E1 12463.018,E2 12463.018} C_VEL
LIN {X 0,Y 406.879,Z 947.579,A -85,B 0,C 180,E1 12461.77,E2 12461.77} C_VEL
LIN {X 0,Y 409.793,Z 927.06,A -85,B 0,C 180,E1 12460.874,E2 12460.874} C_VEL
LIN {X 0,Y 412.466,Z 903.221,A -85,B 0,C 180,E1 12460.09,E2 12460.09} C_VEL
LIN {X 0,Y 414.22,Z 879.631,A -85,B 0,C 180,E1 12459.533,E2 12459.533} C_VEL
LIN {X 0,Y 424.374,Z 670.007,A -85,B 0,C 180,E1 12455.427,E2 12455.427} C_VEL
LIN {X 0,Y 426.37,Z 627.382,A -85,B 0,C 180,E1 12454.576,E2 12454.576} C_VEL
LIN {X 0,Y 415.774,Z 611.035,A -85,B 0,C 180,E1 12452.104,E2 12452.104} C_VEL
LIN {X 0,Y 405.962,Z 597.188,A -85,B 0,C 180,E1 12449.591,E2 12449.591} C_VEL
LIN {X 0,Y 398.176,Z 586.901,A -85,B 0,C 180,E1 12447.397,E2 12447.397} C_VEL
LIN {X 0,Y 393.883,Z 581.421,A -85,B 0,C 180,E1 12446.09,E2 12446.09} C_VEL
LIN {X 0,Y 389.76,Z 576.302,A -85,B 0,C 180,E1 12444.758,E2 12444.758} C_VEL
LIN {X 0,Y 385.613,Z 571.304,A -85,B 0,C 180,E1 12443.332,E2 12443.332} C_VEL
LIN {X 0,Y 381.217,Z 566.1,A -85,B 0,C 180,E1 12441.704,E2 12441.704} C_VEL
LIN {X 0,Y 376.318,Z 560.498,A -85,B 0,C 180,E1 12439.72,E2 12439.72} C_VEL
LIN {X 0,Y 373.744,Z 557.541,A -85,B 0,C 180,E1 12438.401,E2 12438.401} C_VEL
LIN {X 0,Y 372.652,Z 555.125,A -85,B 0,C 180,E1 12437.326,E2 12437.326} C_VEL
LIN {X 0,Y 370.01,Z 551.43,A -85,B 0,C 180,E1 12435.035,E2 12435.035} C_VEL
LIN {X 0,Y 369.088,Z 549.498,A -85,B 0,C 180,E1 12433.951,E2 12433.951} C_VEL
LIN {X 0,Y 366.281,Z 545.751,A -85,B 0,C 180,E1 12430.856,E2 12430.856} C_VEL
LIN {X 0,Y 365.354,Z 543.75,A -85,B 0,C 180,E1 12429.291,E2 12429.291} C_VEL
LIN {X 0,Y 362.092,Z 539.341,A -85,B 0,C 180,E1 12421.898,E2 12421.898} C_VEL
LIN {X 0,Y 361.938,Z 538.749,A -85,B 0,C 180,E1 12418.417,E2 12418.417} C_VEL
LIN {X 0,Y 362.241,Z 539.767,A -85,B 0,C 180,E1 12414.615,E2 12414.615} C_VEL
LIN {X 0,Y 365.737,Z 544.204,A -85,B 0,C 180,E1 12407.687,E2 12407.687} C_VEL
LIN {X 0,Y 368.084,Z 548.604,A -85,B 0,C 180,E1 12404.399,E2 12404.399} C_VEL
LIN {X 0,Y 369.423,Z 550.02,A -85,B 0,C 180,E1 12403.166,E2 12403.166} C_VEL
LIN {X 0,Y 371.642,Z 554.151,A -85,B 0,C 180,E1 12400.838,E2 12400.838} C_VEL
LIN {X 0,Y 372.969,Z 555.918,A -85,B 0,C 180,E1 12399.766,E2 12399.766} C_VEL
LIN {X 0,Y 375.126,Z 559.767,A -85,B 0,C 180,E1 12397.925,E2 12397.925} C_VEL
LIN {X 0,Y 376.167,Z 561.314,A -85,B 0,C 180,E1 12397.165,E2 12397.165} C_VEL
LIN {X 0,Y 378.708,Z 565.485,A -85,B 0,C 180,E1 12395.345,E2 12395.345} C_VEL
LIN {X 0,Y 382.215,Z 572.018,A -85,B 0,C 180,E1 12392.923,E2 12392.923} C_VEL
LIN {X 0,Y 384.982,Z 576.706,A -85,B 0,C 180,E1 12391.368,E2 12391.368} C_VEL
LIN {X 0,Y 392.838,Z 587.263,A -85,B 0,C 180,E1 12388.719,E2 12388.719} C_VEL
LIN {X 0,Y 399.368,Z 596.304,A -85,B 0,C 180,E1 12386.742,E2 12386.742} C_VEL
LIN {X 0,Y 407.989,Z 608.944,A -85,B 0,C 180,E1 12384.362,E2 12384.362} C_VEL
LIN {X 0,Y 418.547,Z 625.484,A -85,B 0,C 180,E1 12381.733,E2 12381.733} C_VEL
LIN {X 0,Y 422.477,Z 632.393,A -85,B 0,C 180,E1 12380.809,E2 12380.809} C_VEL
LIN {X 0,Y 423.034,Z 638.84,A -85,B 0,C 180,E1 12380.536,E2 12380.536} C_VEL
LIN {X 0,Y 413.413,Z 870.933,A -85,B 0,C 180,E1 12376.299,E2 12376.299} C_VEL
LIN {X 0,Y 411.853,Z 901.296,A -85,B 0,C 180,E1 12375.696,E2 12375.696} C_VEL
LIN {X 0,Y 409.75,Z 922.76,A -85,B 0,C 180,E1 12375.075,E2 12375.075} C_VEL
LIN {X 0,Y 406.996,Z 943.314,A -85,B 0,C 180,E1 12374.243,E2 12374.243} C_VEL
LIN {X 0,Y 403.763,Z 963.221,A -85,B 0,C 180,E1 12373.213,E2 12373.213} C_VEL
LIN {X 0,Y 399.976,Z 982.377,A -85,B 0,C 180,E1 12371.967,E2 12371.967} C_VEL
LIN {X 0,Y 395.401,Z 1002.735,A -85,B 0,C 180,E1 12370.343,E2 12370.343} C_VEL
LIN {X 0,Y 390.827,Z 1021.205,A -85,B 0,C 180,E1 12368.555,E2 12368.555} C_VEL
LIN {X 0,Y 386.159,Z 1038.319,A -85,B 0,C 180,E1 12366.55,E2 12366.55} C_VEL
LIN {X 0,Y 381.203,Z 1055.559,A -85,B 0,C 180,E1 12364.146,E2 12364.146} C_VEL
LIN {X 0,Y 376.848,Z 1070.396,A -85,B 0,C 180,E1 12361.691,E2 12361.691} C_VEL
LIN {X 0,Y 372.822,Z 1083.805,A -85,B 0,C 180,E1 12359.038,E2 12359.038} C_VEL
LIN {X 0,Y 369.087,Z 1096.648,A -85,B 0,C 180,E1 12356.031,E2 12356.031} C_VEL
LIN {X 0,Y 366.582,Z 1105.707,A -85,B 0,C 180,E1 12353.531,E2 12353.531} C_VEL
LIN {X 0,Y 364.71,Z 1109.364,A -85,B 0,C 180,E1 12352.497,E2 12352.497} C_VEL
LIN {X 0,Y 356.504,Z 1118.506,A -85,B 0,C 180,E1 12349.739,E2 12349.739} C_VEL
LIN {X 0,Y 355.176,Z 1120.985,A -85,B 0,C 180,E1 12348.766,E2 12348.766} C_VEL
LIN {X 0,Y 353.602,Z 1128.561,A -85,B 0,C 180,E1 12345.246,E2 12345.246} C_VEL
LIN {X 0,Y 352.668,Z 1134.238,A -85,B 0,C 180,E1 12341.779,E2 12341.779} C_VEL
LIN {X 0,Y 352.173,Z 1138.61,A -85,B 0,C 180,E1 12338.161,E2 12338.161} C_VEL
LIN {X 0,Y 351.99,Z 1141.179,A -85,B 0,C 180,E1 12334.889,E2 12334.889} C_VEL
LIN {X 0,Y 351.952,Z 1142.5,A -85,B 0,C 180,E1 12331.302,E2 12331.302} C_VEL
LIN {X 0,Y 351.953,Z 1142.428,A -85,B 0,C 180,E1 12328.046,E2 12328.046} C_VEL
LIN {X 0,Y 352.001,Z 1140.918,A -85,B 0,C 180,E1 12324.621,E2 12324.621} C_VEL
LIN {X 0,Y 352.238,Z 1138.09,A -85,B 0,C 180,E1 12321.183,E2 12321.183} C_VEL
LIN {X 0,Y 352.744,Z 1133.65,A -85,B 0,C 180,E1 12317.726,E2 12317.726} C_VEL
LIN {X 0,Y 353.804,Z 1127.41,A -85,B 0,C 180,E1 12314.09,E2 12314.09} C_VEL
LIN {X 0,Y 355.489,Z 1119.759,A -85,B 0,C 180,E1 12310.616,E2 12310.616} C_VEL
LIN {X 0,Y 357.896,Z 1110.341,A -85,B 0,C 180,E1 12307.21,E2 12307.21} C_VEL
LIN {X 0,Y 361.272,Z 1098.606,A -85,B 0,C 180,E1 12303.729,E2 12303.729} C_VEL
LIN {X 0,Y 364.921,Z 1086.812,A -85,B 0,C 180,E1 12300.81,E2 12300.81} C_VEL
LIN {X 0,Y 369.277,Z 1072.826,A -85,B 0,C 180,E1 12297.939,E2 12297.939} C_VEL
LIN {X 0,Y 374.053,Z 1057.488,A -85,B 0,C 180,E1 12295.294,E2 12295.294} C_VEL
LIN {X 0,Y 378.867,Z 1041.78,A -85,B 0,C 180,E1 12293.007,E2 12293.007} C_VEL
LIN {X 0,Y 383.778,Z 1024.496,A -85,B 0,C 180,E1 12290.914,E2 12290.914} C_VEL
LIN {X 0,Y 388.736,Z 1005.715,A -85,B 0,C 180,E1 12289.013,E2 12289.013} C_VEL
LIN {X 0,Y 393.265,Z 987.001,A -85,B 0,C 180,E1 12287.445,E2 12287.445} C_VEL
LIN {X 0,Y 397.35,Z 967.335,A -85,B 0,C 180,E1 12286.112,E2 12286.112} C_VEL
LIN {X 0,Y 401.165,Z 945.76,A -85,B 0,C 180,E1 12284.94,E2 12284.94} C_VEL
LIN {X 0,Y 404.118,Z 925.124,A -85,B 0,C 180,E1 12284.074,E2 12284.074} C_VEL
LIN {X 0,Y 406.393,Z 903.354,A -85,B 0,C 180,E1 12283.42,E2 12283.42} C_VEL
LIN {X 0,Y 408.038,Z 875.14,A -85,B 0,C 180,E1 12282.837,E2 12282.837} C_VEL
LIN {X 0,Y 417.294,Z 660.372,A -85,B 0,C 180,E1 12278.886,E2 12278.886} C_VEL
LIN {X 0,Y 411.931,Z 666.042,A -85,B 0,C 180,E1 12278.019,E2 12278.019} C_VEL
LIN {X 0,Y 406.165,Z 674.715,A -85,B 0,C 180,E1 12277.116,E2 12277.116} C_VEL
LIN {X 0,Y 401.389,Z 679.876,A -85,B 0,C 180,E1 12276.272,E2 12276.272} C_VEL
LIN {X 0,Y 395.378,Z 689.653,A -85,B 0,C 180,E1 12275.255,E2 12275.255} C_VEL
LIN {X 0,Y 391.308,Z 694.358,A -85,B 0,C 180,E1 12274.47,E2 12274.47} C_VEL
LIN {X 0,Y 390.198,Z 695.593,A -85,B 0,C 180,E1 12274.248,E2 12274.248} C_VEL
LIN {X 0,Y 385.36,Z 704.501,A -85,B 0,C 180,E1 12273.371,E2 12273.371} C_VEL
LIN {X 0,Y 381.697,Z 709.399,A -85,B 0,C 180,E1 12272.614,E2 12272.614} C_VEL
LIN {X 0,Y 379.74,Z 711.492,A -85,B 0,C 180,E1 12272.177,E2 12272.177} C_VEL
LIN {X 0,Y 374.529,Z 722.032,A -85,B 0,C 180,E1 12271.148,E2 12271.148} C_VEL
LIN {X 0,Y 371.463,Z 726.494,A -85,B 0,C 180,E1 12270.445,E2 12270.445} C_VEL
LIN {X 0,Y 370.055,Z 728.582,A -85,B 0,C 180,E1 12269.991,E2 12269.991} C_VEL
LIN {X 0,Y 370.127,Z 733.475,A -85,B 0,C 180,E1 12269.695,E2 12269.695} C_VEL
LIN {X 0,Y 364.868,Z 900.694,A -85,B 0,C 180,E1 12265.755,E2 12265.755} C_VEL
LIN {X 0,Y 364.266,Z 918.714,A -85,B 0,C 180,E1 12265.054,E2 12265.054} C_VEL
LIN {X 0,Y 363.315,Z 936.828,A -85,B 0,C 180,E1 12264.036,E2 12264.036} C_VEL
LIN {X 0,Y 362.191,Z 953.289,A -85,B 0,C 180,E1 12262.813,E2 12262.813} C_VEL
LIN {X 0,Y 360.868,Z 969.289,A -85,B 0,C 180,E1 12261.283,E2 12261.283} C_VEL
LIN {X 0,Y 359.469,Z 984.283,A -85,B 0,C 180,E1 12259.499,E2 12259.499} C_VEL
LIN {X 0,Y 358.137,Z 997.484,A -85,B 0,C 180,E1 12257.549,E2 12257.549} C_VEL
LIN {X 0,Y 356.853,Z 1009.96,A -85,B 0,C 180,E1 12255.271,E2 12255.271} C_VEL
LIN {X 0,Y 355.868,Z 1020.044,A -85,B 0,C 180,E1 12252.99,E2 12252.99} C_VEL
LIN {X 0,Y 355.077,Z 1028.595,A -85,B 0,C 180,E1 12250.547,E2 12250.547} C_VEL
LIN {X 0,Y 354.537,Z 1035.679,A -85,B 0,C 180,E1 12247.943,E2 12247.943} C_VEL
LIN {X 0,Y 354.258,Z 1040.873,A -85,B 0,C 180,E1 12245.345,E2 12245.345} C_VEL
LIN {X 0,Y 354.174,Z 1044.284,A -85,B 0,C 180,E1 12242.751,E2 12242.751} C_VEL
LIN {X 0,Y 354.266,Z 1046.163,A -85,B 0,C 180,E1 12240,E2 12240} C_VEL
LIN {X 0,Y 354.493,Z 1046.277,A -85,B 0,C 180,E1 12237.414,E2 12237.414} C_VEL
LIN {X 0,Y 354.873,Z 1044.713,A -85,B 0,C 180,E1 12234.828,E2 12234.828} C_VEL
LIN {X 0,Y 355.465,Z 1041.437,A -85,B 0,C 180,E1 12232.241,E2 12232.241} C_VEL
LIN {X 0,Y 356.322,Z 1036.342,A -85,B 0,C 180,E1 12229.655,E2 12229.655} C_VEL
LIN {X 0,Y 357.38,Z 1029.695,A -85,B 0,C 180,E1 12227.231,E2 12227.231} C_VEL
LIN {X 0,Y 358.577,Z 1021.518,A -85,B 0,C 180,E1 12224.971,E2 12224.971} C_VEL
LIN {X 0,Y 359.931,Z 1011.917,A -85,B 0,C 180,E1 12222.864,E2 12222.864} C_VEL
LIN {X 0,Y 361.337,Z 1000.985,A -85,B 0,C 180,E1 12220.943,E2 12220.943} C_VEL
LIN {X 0,Y 362.797,Z 987.951,A -85,B 0,C 180,E1 12219.112,E2 12219.112} C_VEL
LIN {X 0,Y 364.093,Z 974.168,A -85,B 0,C 180,E1 12217.56,E2 12217.56} C_VEL
LIN {X 0,Y 365.237,Z 958.752,A -85,B 0,C 180,E1 12216.185,E2 12216.185} C_VEL
LIN {X 0,Y 366.17,Z 941.915,A -85,B 0,C 180,E1 12215.034,E2 12215.034} C_VEL
LIN {X 0,Y 366.765,Z 924.329,A -85,B 0,C 180,E1 12214.156,E2 12214.156} C_VEL
LIN {X 0,Y 367.092,Z 903.612,A -85,B 0,C 180,E1 12213.464,E2 12213.464} C_VEL
LIN {X 0,Y 369.766,Z 843.304,A -85,B 0,C 180,E1 12211.791,E2 12211.791} C_VEL
LIN {X 0,Y 371.625,Z 816.569,A -85,B 0,C 180,E1 12210.977,E2 12210.977} C_VEL
LIN {X 0,Y 373.015,Z 810.856,A -85,B 0,C 180,E1 12210.658,E2 12210.658} C_VEL
LIN {X 0,Y 376.424,Z 801.259,A -85,B 0,C 180,E1 12210.163,E2 12210.163} C_VEL
LIN {X 0,Y 381.337,Z 783.402,A -85,B 0,C 180,E1 12209.639,E2 12209.639} C_VEL
LIN {X 0,Y 384.822,Z 770.175,A -85,B 0,C 180,E1 12209.3,E2 12209.3} C_VEL
LIN {X 0,Y 389.205,Z 758.51,A -85,B 0,C 180,E1 12208.718,E2 12208.718} C_VEL
LIN {X 0,Y 391.128,Z 753.356,A -85,B 0,C 180,E1 12208.471,E2 12208.471} C_VEL
LIN {X 0,Y 396.162,Z 742.423,A -85,B 0,C 180,E1 12207.76,E2 12207.76} C_VEL
LIN {X 0,Y 401.216,Z 736.224,A -85,B 0,C 180,E1 12206.924,E2 12206.924} C_VEL
LIN {X 0,Y 406.728,Z 727.21,A -85,B 0,C 180,E1 12206.123,E2 12206.123} C_VEL
LIN {X 0,Y 411.911,Z 720.836,A -85,B 0,C 180,E1 12205.343,E2 12205.343} C_VEL
LIN {X 0,Y 416.797,Z 713.303,A -85,B 0,C 180,E1 12204.681,E2 12204.681} C_VEL
LIN {X 0,Y 417.295,Z 712.94,A -85,B 0,C 180,E1 12204.603,E2 12204.603} C_VEL
LIN {X 0,Y 408.175,Z 891.531,A -85,B 0,C 180,E1 12201.048,E2 12201.048} C_VEL
LIN {X 0,Y 405.821,Z 915.215,A -85,B 0,C 180,E1 12200.387,E2 12200.387} C_VEL
LIN {X 0,Y 402.991,Z 937.031,A -85,B 0,C 180,E1 12199.559,E2 12199.559} C_VEL
LIN {X 0,Y 399.372,Z 958.94,A -85,B 0,C 180,E1 12198.467,E2 12198.467} C_VEL
LIN {X 0,Y 395.2,Z 980.794,A -85,B 0,C 180,E1 12197.112,E2 12197.112} C_VEL
LIN {X 0,Y 390.959,Z 1000.382,A -85,B 0,C 180,E1 12195.628,E2 12195.628} C_VEL
LIN {X 0,Y 385.95,Z 1021.372,A -85,B 0,C 180,E1 12193.715,E2 12193.715} C_VEL
LIN {X 0,Y 381.201,Z 1039.966,A -85,B 0,C 180,E1 12191.709,E2 12191.709} C_VEL
LIN {X 0,Y 376.33,Z 1057.831,A -85,B 0,C 180,E1 12189.42,E2 12189.42} C_VEL
LIN {X 0,Y 371.545,Z 1075.242,A -85,B 0,C 180,E1 12186.814,E2 12186.814} C_VEL
LIN {X 0,Y 367.256,Z 1090.575,A -85,B 0,C 180,E1 12184.114,E2 12184.114} C_VEL
LIN {X 0,Y 363.151,Z 1105.751,A -85,B 0,C 180,E1 12180.989,E2 12180.989} C_VEL
LIN {X 0,Y 359.796,Z 1118.844,A -85,B 0,C 180,E1 12177.831,E2 12177.831} C_VEL
LIN {X 0,Y 357.018,Z 1130.561,A -85,B 0,C 180,E1 12174.47,E2 12174.47} C_VEL
LIN {X 0,Y 354.997,Z 1140.496,A -85,B 0,C 180,E1 12171.132,E2 12171.132} C_VEL
LIN {X 0,Y 353.52,Z 1149.027,A -85,B 0,C 180,E1 12167.613,E2 12167.613} C_VEL
LIN {X 0,Y 352.622,Z 1155.997,A -85,B 0,C 180,E1 12164.114,E2 12164.114} C_VEL
LIN {X 0,Y 352.17,Z 1161.041,A -85,B 0,C 180,E1 12160.787,E2 12160.787} C_VEL
LIN {X 0,Y 351.964,Z 1164.773,A -85,B 0,C 180,E1 12157.507,E2 12157.507} C_VEL
LIN {X 0,Y 351.932,Z 1167.257,A -85,B 0,C 180,E1 12153.91,E2 12153.91} C_VEL
LIN {X 0,Y 351.922,Z 1168.134,A -85,B 0,C 180,E1 12150.977,E2 12150.977} C_VEL
LIN {X 0,Y 351.932,Z 1167.9,A -85,B 0,C 180,E1 12147.558,E2 12147.558} C_VEL
LIN {X 0,Y 351.931,Z 1166.194,A -85,B 0,C 180,E1 12144.293,E2 12144.293} C_VEL
LIN {X 0,Y 352.041,Z 1163.424,A -85,B 0,C 180,E1 12141.178,E2 12141.178} C_VEL
LIN {X 0,Y 352.371,Z 1158.52,A -85,B 0,C 180,E1 12137.447,E2 12137.447} C_VEL
LIN {X 0,Y 352.993,Z 1152.851,A -85,B 0,C 180,E1 12134.221,E2 12134.221} C_VEL
LIN {X 0,Y 354.301,Z 1144.327,A -85,B 0,C 180,E1 12130.377,E2 12130.377} C_VEL
LIN {X 0,Y 356.048,Z 1135.222,A -85,B 0,C 180,E1 12127.024,E2 12127.024} C_VEL
LIN {X 0,Y 358.46,Z 1124.302,A -85,B 0,C 180,E1 12123.672,E2 12123.672} C_VEL
LIN {X 0,Y 361.654,Z 1111.558,A -85,B 0,C 180,E1 12120.338,E2 12120.338} C_VEL
LIN {X 0,Y 365.435,Z 1097.226,A -85,B 0,C 180,E1 12117.197,E2 12117.197} C_VEL
LIN {X 0,Y 370.002,Z 1080.64,A -85,B 0,C 180,E1 12114.098,E2 12114.098} C_VEL
LIN {X 0,Y 374.513,Z 1064.538,A -85,B 0,C 180,E1 12111.534,E2 12111.534} C_VEL
LIN {X 0,Y 379.406,Z 1046.444,A -85,B 0,C 180,E1 12109.089,E2 12109.089} C_VEL
LIN {X 0,Y 384.348,Z 1027.714,A -85,B 0,C 180,E1 12106.931,E2 12106.931} C_VEL
LIN {X 0,Y 388.891,Z 1009.141,A -85,B 0,C 180,E1 12105.133,E2 12105.133} C_VEL
LIN {X 0,Y 393.672,Z 988.069,A -85,B 0,C 180,E1 12103.415,E2 12103.415} C_VEL
LIN {X 0,Y 397.585,Z 968.663,A -85,B 0,C 180,E1 12102.108,E2 12102.108} C_VEL
LIN {X 0,Y 401.48,Z 946.376,A -85,B 0,C 180,E1 12100.885,E2 12100.885} C_VEL
LIN {X 0,Y 404.56,Z 925.35,A -85,B 0,C 180,E1 12099.975,E2 12099.975} C_VEL
LIN {X 0,Y 407.199,Z 902.001,A -85,B 0,C 180,E1 12099.222,E2 12099.222} C_VEL
LIN {X 0,Y 408.99,Z 877.845,A -85,B 0,C 180,E1 12098.661,E2 12098.661} C_VEL
LIN {X 0,Y 419.555,Z 668.638,A -85,B 0,C 180,E1 12094.536,E2 12094.536} C_VEL
LIN {X 0,Y 421.377,Z 631.434,A -85,B 0,C 180,E1 12093.788,E2 12093.788} C_VEL
LIN {X 0,Y 411.551,Z 616.162,A -85,B 0,C 180,E1 12091.407,E2 12091.407} C_VEL
LIN {X 0,Y 402.405,Z 603.126,A -85,B 0,C 180,E1 12088.98,E2 12088.98} C_VEL
LIN {X 0,Y 394.991,Z 593.213,A -85,B 0,C 180,E1 12086.821,E2 12086.821} C_VEL
LIN {X 0,Y 388.365,Z 584.53,A -85,B 0,C 180,E1 12084.69,E2 12084.69} C_VEL
LIN {X 0,Y 382.793,Z 577.916,A -85,B 0,C 180,E1 12082.741,E2 12082.741} C_VEL
LIN {X 0,Y 379.136,Z 573.447,A -85,B 0,C 180,E1 12081.341,E2 12081.341} C_VEL
LIN {X 0,Y 374.317,Z 567.881,A -85,B 0,C 180,E1 12079.343,E2 12079.343} C_VEL
LIN {X 0,Y 369.149,Z 562.075,A -85,B 0,C 180,E1 12076.927,E2 12076.927} C_VEL
LIN {X 0,Y 366.392,Z 559.162,A -85,B 0,C 180,E1 12075.349,E2 12075.349} C_VEL
LIN {X 0,Y 365.06,Z 556.358,A -85,B 0,C 180,E1 12073.785,E2 12073.785} C_VEL
LIN {X 0,Y 362.326,Z 552.585,A -85,B 0,C 180,E1 12070.654,E2 12070.654} C_VEL
LIN {X 0,Y 361.519,Z 550.761,A -85,B 0,C 180,E1 12069.23,E2 12069.23} C_VEL
LIN {X 0,Y 358.319,Z 546.408,A -85,B 0,C 180,E1 12061.918,E2 12061.918} C_VEL
LIN {X 0,Y 358.11,Z 545.782,A -85,B 0,C 180,E1 12058.292,E2 12058.292} C_VEL
LIN {X 0,Y 358.48,Z 546.868,A -85,B 0,C 180,E1 12054.558,E2 12054.558} C_VEL
LIN {X 0,Y 361.781,Z 551.063,A -85,B 0,C 180,E1 12047.875,E2 12047.875} C_VEL
LIN {X 0,Y 364.218,Z 555.627,A -85,B 0,C 180,E1 12044.393,E2 12044.393} C_VEL
LIN {X 0,Y 365.354,Z 556.916,A -85,B 0,C 180,E1 12043.3,E2 12043.3} C_VEL
LIN {X 0,Y 367.565,Z 560.999,A -85,B 0,C 180,E1 12040.948,E2 12040.948} C_VEL
LIN {X 0,Y 368.693,Z 562.486,A -85,B 0,C 180,E1 12040.019,E2 12040.019} C_VEL
LIN {X 0,Y 370.79,Z 566.36,A -85,B 0,C 180,E1 12038.153,E2 12038.153} C_VEL
LIN {X 0,Y 371.816,Z 567.897,A -85,B 0,C 180,E1 12037.384,E2 12037.384} C_VEL
LIN {X 0,Y 374.881,Z 573.376,A -85,B 0,C 180,E1 12035.071,E2 12035.071} C_VEL
LIN {X 0,Y 377.767,Z 577.342,A -85,B 0,C 180,E1 12033.683,E2 12033.683} C_VEL
LIN {X 0,Y 383.165,Z 584.584,A -85,B 0,C 180,E1 12031.603,E2 12031.603} C_VEL
LIN {X 0,Y 390.12,Z 594.014,A -85,B 0,C 180,E1 12029.206,E2 12029.206} C_VEL
LIN {X 0,Y 396.845,Z 603.503,A -85,B 0,C 180,E1 12027.115,E2 12027.115} C_VEL
LIN {X 0,Y 405.61,Z 616.63,A -85,B 0,C 180,E1 12024.642,E2 12024.642} C_VEL
LIN {X 0,Y 415.374,Z 632.256,A -85,B 0,C 180,E1 12022.155,E2 12022.155} C_VEL
LIN {X 0,Y 417.991,Z 637.053,A -85,B 0,C 180,E1 12021.518,E2 12021.518} C_VEL
LIN {X 0,Y 418.166,Z 641.035,A -85,B 0,C 180,E1 12021.375,E2 12021.375} C_VEL
LIN {X 0,Y 408.089,Z 872.811,A -85,B 0,C 180,E1 12017.11,E2 12017.11} C_VEL
LIN {X 0,Y 406.451,Z 902.214,A -85,B 0,C 180,E1 12016.514,E2 12016.514} C_VEL
LIN {X 0,Y 404.207,Z 924.119,A -85,B 0,C 180,E1 12015.868,E2 12015.868} C_VEL
LIN {X 0,Y 401.345,Z 944.284,A -85,B 0,C 180,E1 12015.034,E2 12015.034} C_VEL
LIN {X 0,Y 397.762,Z 965.09,A -85,B 0,C 180,E1 12013.931,E2 12013.931} C_VEL
LIN {X 0,Y 393.856,Z 984.045,A -85,B 0,C 180,E1 12012.673,E2 12012.673} C_VEL
LIN {X 0,Y 389.313,Z 1003.302,A -85,B 0,C 180,E1 12011.108,E2 12011.108} C_VEL
LIN {X 0,Y 384.69,Z 1021.201,A -85,B 0,C 180,E1 12009.36,E2 12009.36} C_VEL
LIN {X 0,Y 379.68,Z 1038.79,A -85,B 0,C 180,E1 12007.279,E2 12007.279} C_VEL
LIN {X 0,Y 374.655,Z 1055.493,A -85,B 0,C 180,E1 12004.921,E2 12004.921} C_VEL
LIN {X 0,Y 369.926,Z 1070.792,A -85,B 0,C 180,E1 12002.355,E2 12002.355} C_VEL
LIN {X 0,Y 365.565,Z 1084.619,A -85,B 0,C 180,E1 11999.568,E2 11999.568} C_VEL
LIN {X 0,Y 361.56,Z 1097.623,A -85,B 0,C 180,E1 11996.438,E2 11996.438} C_VEL
LIN {X 0,Y 358.443,Z 1108.424,A -85,B 0,C 180,E1 11993.335,E2 11993.335} C_VEL
LIN {X 0,Y 355.94,Z 1117.814,A -85,B 0,C 180,E1 11990.042,E2 11990.042} C_VEL
LIN {X 0,Y 355.176,Z 1120.985,A -85,B 0,C 180,E1 11988.766,E2 11988.766} C_VEL
LIN {X 0,Y 353.585,Z 1123.836,A -85,B 0,C 180,E1 11987.621,E2 11987.621} C_VEL
LIN {X 0,Y 346.143,Z 1130.596,A -85,B 0,C 180,E1 11984.555,E2 11984.555} C_VEL
LIN {X 0,Y 345.082,Z 1132.447,A -85,B 0,C 180,E1 11983.507,E2 11983.507} C_VEL
LIN {X 0,Y 344.384,Z 1137.121,A -85,B 0,C 180,E1 11980.032,E2 11980.032} C_VEL
LIN {X 0,Y 344.08,Z 1140.511,A -85,B 0,C 180,E1 11976.507,E2 11976.507} C_VEL
LIN {X 0,Y 343.966,Z 1142.313,A -85,B 0,C 180,E1 11973.166,E2 11973.166} C_VEL
LIN {X 0,Y 343.953,Z 1142.932,A -85,B 0,C 180,E1 11969.667,E2 11969.667} C_VEL
LIN {X 0,Y 343.976,Z 1142.158,A -85,B 0,C 180,E1 11966.333,E2 11966.333} C_VEL
LIN {X 0,Y 344.112,Z 1139.898,A -85,B 0,C 180,E1 11962.655,E2 11962.655} C_VEL
LIN {X 0,Y 344.469,Z 1136.448,A -85,B 0,C 180,E1 11959.294,E2 11959.294} C_VEL
LIN {X 0,Y 345.326,Z 1131.056,A -85,B 0,C 180,E1 11955.581,E2 11955.581} C_VEL
LIN {X 0,Y 346.757,Z 1124.338,A -85,B 0,C 180,E1 11952.029,E2 11952.029} C_VEL
LIN {X 0,Y 348.929,Z 1115.748,A -85,B 0,C 180,E1 11948.482,E2 11948.482} C_VEL
LIN {X 0,Y 351.984,Z 1105.256,A -85,B 0,C 180,E1 11944.96,E2 11944.96} C_VEL
LIN {X 0,Y 355.574,Z 1093.949,A -85,B 0,C 180,E1 11941.809,E2 11941.809} C_VEL
LIN {X 0,Y 359.728,Z 1081.227,A -85,B 0,C 180,E1 11938.87,E2 11938.87} C_VEL
LIN {X 0,Y 364.356,Z 1067.214,A -85,B 0,C 180,E1 11936.146,E2 11936.146} C_VEL
LIN {X 0,Y 369.345,Z 1051.966,A -85,B 0,C 180,E1 11933.64,E2 11933.64} C_VEL
LIN {X 0,Y 374.546,Z 1035.107,A -85,B 0,C 180,E1 11931.342,E2 11931.342} C_VEL
LIN {X 0,Y 379.878,Z 1016.72,A -85,B 0,C 180,E1 11929.251,E2 11929.251} C_VEL
LIN {X 0,Y 384.824,Z 998.243,A -85,B 0,C 180,E1 11927.504,E2 11927.504} C_VEL
LIN {X 0,Y 389.367,Z 978.752,A -85,B 0,C 180,E1 11926.003,E2 11926.003} C_VEL
LIN {X 0,Y 393.703,Z 957.349,A -85,B 0,C 180,E1 11924.676,E2 11924.676} C_VEL
LIN {X 0,Y 397.249,Z 936.33,A -85,B 0,C 180,E1 11923.652,E2 11923.652} C_VEL
LIN {X 0,Y 399.912,Z 915.739,A -85,B 0,C 180,E1 11922.905,E2 11922.905} C_VEL
LIN {X 0,Y 402.019,Z 892.352,A -85,B 0,C 180,E1 11922.306,E2 11922.306} C_VEL
LIN {X 0,Y 411.817,Z 676.228,A -85,B 0,C 180,E1 11918.282,E2 11918.282} C_VEL
LIN {X 0,Y 406.434,Z 683.304,A -85,B 0,C 180,E1 11917.419,E2 11917.419} C_VEL
LIN {X 0,Y 403.103,Z 686.968,A -85,B 0,C 180,E1 11916.844,E2 11916.844} C_VEL
LIN {X 0,Y 397.854,Z 695.377,A -85,B 0,C 180,E1 11915.981,E2 11915.981} C_VEL
LIN {X 0,Y 393.226,Z 700.809,A -85,B 0,C 180,E1 11915.12,E2 11915.12} C_VEL
LIN {X 0,Y 392.138,Z 702.327,A -85,B 0,C 180,E1 11914.92,E2 11914.92} C_VEL
LIN {X 0,Y 387.117,Z 711.064,A -85,B 0,C 180,E1 11914.022,E2 11914.022} C_VEL
LIN {X 0,Y 383.047,Z 716.258,A -85,B 0,C 180,E1 11913.196,E2 11913.196} C_VEL
LIN {X 0,Y 381.676,Z 717.886,A -85,B 0,C 180,E1 11912.906,E2 11912.906} C_VEL
LIN {X 0,Y 376.777,Z 727.523,A -85,B 0,C 180,E1 11911.966,E2 11911.966} C_VEL
LIN {X 0,Y 373.207,Z 732.748,A -85,B 0,C 180,E1 11911.181,E2 11911.181} C_VEL
LIN {X 0,Y 371.999,Z 734.325,A -85,B 0,C 180,E1 11910.9,E2 11910.9} C_VEL
LIN {X 0,Y 366.686,Z 758.117,A -85,B 0,C 180,E1 11910.284,E2 11910.284} C_VEL
LIN {X 0,Y 363.659,Z 768.731,A -85,B 0,C 180,E1 11909.8,E2 11909.8} C_VEL
LIN {X 0,Y 361.842,Z 774.888,A -85,B 0,C 180,E1 11909.361,E2 11909.361} C_VEL
LIN {X 0,Y 361.006,Z 785.636,A -85,B 0,C 180,E1 11908.981,E2 11908.981} C_VEL
LIN {X 0,Y 357.34,Z 901.528,A -85,B 0,C 180,E1 11906.171,E2 11906.171} C_VEL
LIN {X 0,Y 356.715,Z 919.752,A -85,B 0,C 180,E1 11905.45,E2 11905.45} C_VEL
LIN {X 0,Y 355.723,Z 937.992,A -85,B 0,C 180,E1 11904.405,E2 11904.405} C_VEL
LIN {X 0,Y 354.578,Z 954.232,A -85,B 0,C 180,E1 11903.179,E2 11903.179} C_VEL
LIN {X 0,Y 353.258,Z 969.773,A -85,B 0,C 180,E1 11901.677,E2 11901.677} C_VEL
LIN {X 0,Y 351.865,Z 984.306,A -85,B 0,C 180,E1 11899.938,E2 11899.938} C_VEL
LIN {X 0,Y 350.475,Z 997.847,A -85,B 0,C 180,E1 11897.946,E2 11897.946} C_VEL
LIN {X 0,Y 349.206,Z 1009.706,A -85,B 0,C 180,E1 11895.784,E2 11895.784} C_VEL
LIN {X 0,Y 348.146,Z 1020.139,A -85,B 0,C 180,E1 11893.452,E2 11893.452} C_VEL
LIN {X 0,Y 347.3,Z 1029.054,A -85,B 0,C 180,E1 11890.954,E2 11890.954} C_VEL
LIN {X 0,Y 346.703,Z 1036.383,A -85,B 0,C 180,E1 11888.291,E2 11888.291} C_VEL
LIN {X 0,Y 346.394,Z 1041.831,A -85,B 0,C 180,E1 11885.633,E2 11885.633} C_VEL
LIN {X 0,Y 346.303,Z 1045.492,A -85,B 0,C 180,E1 11882.979,E2 11882.979} C_VEL
LIN {X 0,Y 346.392,Z 1047.547,A -85,B 0,C 180,E1 11880.166,E2 11880.166} C_VEL
LIN {X 0,Y 346.628,Z 1047.847,A -85,B 0,C 180,E1 11877.521,E2 11877.521} C_VEL
LIN {X 0,Y 347.042,Z 1046.503,A -85,B 0,C 180,E1 11874.876,E2 11874.876} C_VEL
LIN {X 0,Y 347.672,Z 1043.41,A -85,B 0,C 180,E1 11872.232,E2 11872.232} C_VEL
LIN {X 0,Y 348.581,Z 1038.488,A -85,B 0,C 180,E1 11869.59,E2 11869.59} C_VEL
LIN {X 0,Y 349.702,Z 1032.027,A -85,B 0,C 180,E1 11867.114,E2 11867.114} C_VEL
LIN {X 0,Y 350.984,Z 1024.096,A -85,B 0,C 180,E1 11864.807,E2 11864.807} C_VEL
LIN {X 0,Y 352.39,Z 1014.71,A -85,B 0,C 180,E1 11862.668,E2 11862.668} C_VEL
LIN {X 0,Y 353.918,Z 1003.793,A -85,B 0,C 180,E1 11860.664,E2 11860.664} C_VEL
LIN {X 0,Y 355.388,Z 991.793,A -85,B 0,C 180,E1 11858.893,E2 11858.893} C_VEL
LIN {X 0,Y 356.875,Z 977.331,A -85,B 0,C 180,E1 11857.186,E2 11857.186} C_VEL
LIN {X 0,Y 358.115,Z 962.152,A -85,B 0,C 180,E1 11855.769,E2 11855.769} C_VEL
LIN {X 0,Y 359.151,Z 945.472,A -85,B 0,C 180,E1 11854.57,E2 11854.57} C_VEL
LIN {X 0,Y 359.837,Z 928.235,A -85,B 0,C 180,E1 11853.648,E2 11853.648} C_VEL
LIN {X 0,Y 360.253,Z 907.102,A -85,B 0,C 180,E1 11852.886,E2 11852.886} C_VEL
LIN {X 0,Y 362.184,Z 865.348,A -85,B 0,C 180,E1 11851.647,E2 11851.647} C_VEL
LIN {X 0,Y 363.429,Z 858.396,A -85,B 0,C 180,E1 11851.299,E2 11851.299} C_VEL
LIN {X 0,Y 366.705,Z 849.36,A -85,B 0,C 180,E1 11850.776,E2 11850.776} C_VEL
LIN {X 0,Y 371.447,Z 832.38,A -85,B 0,C 180,E1 11850.228,E2 11850.228} C_VEL
LIN {X 0,Y 375.426,Z 816.85,A -85,B 0,C 180,E1 11849.833,E2 11849.833} C_VEL
LIN {X 0,Y 379.696,Z 805.503,A -85,B 0,C 180,E1 11849.235,E2 11849.235} C_VEL
LIN {X 0,Y 384.611,Z 788.345,A -85,B 0,C 180,E1 11848.716,E2 11848.716} C_VEL
LIN {X 0,Y 388.658,Z 773.03,A -85,B 0,C 180,E1 11848.345,E2 11848.345} C_VEL
LIN {X 0,Y 392.955,Z 761.775,A -85,B 0,C 180,E1 11847.799,E2 11847.799} C_VEL
LIN {X 0,Y 394.943,Z 756.597,A -85,B 0,C 180,E1 11847.551,E2 11847.551} C_VEL
LIN {X 0,Y 398.934,Z 747.972,A -85,B 0,C 180,E1 11847.01,E2 11847.01} C_VEL
LIN {X 0,Y 403.899,Z 741.892,A -85,B 0,C 180,E1 11846.217,E2 11846.217} C_VEL
LIN {X 0,Y 409.557,Z 732.919,A -85,B 0,C 180,E1 11845.417,E2 11845.417} C_VEL
LIN {X 0,Y 411.46,Z 730.973,A -85,B 0,C 180,E1 11845.125,E2 11845.125} C_VEL
LIN {X 0,Y 402.914,Z 891.768,A -85,B 0,C 180,E1 11841.9,E2 11841.9} C_VEL
LIN {X 0,Y 400.49,Z 915.324,A -85,B 0,C 180,E1 11841.238,E2 11841.238} C_VEL
LIN {X 0,Y 397.481,Z 937.575,A -85,B 0,C 180,E1 11840.387,E2 11840.387} C_VEL
LIN {X 0,Y 393.713,Z 959.526,A -85,B 0,C 180,E1 11839.283,E2 11839.283} C_VEL
LIN {X 0,Y 389.134,Z 982.357,A -85,B 0,C 180,E1 11837.841,E2 11837.841} C_VEL
LIN {X 0,Y 384.429,Z 1003.208,A -85,B 0,C 180,E1 11836.225,E2 11836.225} C_VEL
LIN {X 0,Y 379.48,Z 1022.718,A -85,B 0,C 180,E1 11834.391,E2 11834.391} C_VEL
LIN {X 0,Y 374.366,Z 1041.734,A -85,B 0,C 180,E1 11832.285,E2 11832.285} C_VEL
LIN {X 0,Y 369.24,Z 1059.649,A -85,B 0,C 180,E1 11829.924,E2 11829.924} C_VEL
LIN {X 0,Y 364.077,Z 1077.361,A -85,B 0,C 180,E1 11827.17,E2 11827.17} C_VEL
LIN {X 0,Y 359.494,Z 1093.09,A -85,B 0,C 180,E1 11824.307,E2 11824.307} C_VEL
LIN {X 0,Y 355.347,Z 1107.539,A -85,B 0,C 180,E1 11821.18,E2 11821.18} C_VEL
LIN {X 0,Y 351.737,Z 1120.934,A -85,B 0,C 180,E1 11817.788,E2 11817.788} C_VEL
LIN {X 0,Y 349.058,Z 1131.751,A -85,B 0,C 180,E1 11814.541,E2 11814.541} C_VEL
LIN {X 0,Y 346.805,Z 1142.273,A -85,B 0,C 180,E1 11810.77,E2 11810.77} C_VEL
LIN {X 0,Y 345.437,Z 1150.157,A -85,B 0,C 180,E1 11807.345,E2 11807.345} C_VEL
LIN {X 0,Y 344.524,Z 1157.007,A -85,B 0,C 180,E1 11803.596,E2 11803.596} C_VEL
LIN {X 0,Y 344.12,Z 1161.573,A -85,B 0,C 180,E1 11800.378,E2 11800.378} C_VEL
LIN {X 0,Y 343.962,Z 1165.289,A -85,B 0,C 180,E1 11796.677,E2 11796.677} C_VEL
LIN {X 0,Y 343.922,Z 1167.177,A -85,B 0,C 180,E1 11793.5,E2 11793.5} C_VEL
LIN {X 0,Y 343.935,Z 1167.961,A -85,B 0,C 180,E1 11790.167,E2 11790.167} C_VEL
LIN {X 0,Y 343.919,Z 1167.248,A -85,B 0,C 180,E1 11786.667,E2 11786.667} C_VEL
LIN {X 0,Y 343.956,Z 1165.53,A -85,B 0,C 180,E1 11783.658,E2 11783.658} C_VEL
LIN {X 0,Y 344.083,Z 1162.175,A -85,B 0,C 180,E1 11780.089,E2 11780.089} C_VEL
LIN {X 0,Y 344.464,Z 1157.543,A -85,B 0,C 180,E1 11776.744,E2 11776.744} C_VEL
LIN {X 0,Y 345.289,Z 1151.234,A -85,B 0,C 180,E1 11773.168,E2 11773.168} C_VEL
LIN {X 0,Y 346.65,Z 1143.12,A -85,B 0,C 180,E1 11769.573,E2 11769.573} C_VEL
LIN {X 0,Y 348.713,Z 1133.364,A -85,B 0,C 180,E1 11765.974,E2 11765.974} C_VEL
LIN {X 0,Y 351.422,Z 1122.126,A -85,B 0,C 180,E1 11762.553,E2 11762.553} C_VEL
LIN {X 0,Y 355.145,Z 1108.254,A -85,B 0,C 180,E1 11758.988,E2 11758.988} C_VEL
LIN {X 0,Y 359.094,Z 1094.419,A -85,B 0,C 180,E1 11755.967,E2 11755.967} C_VEL
LIN {X 0,Y 363.647,Z 1078.768,A -85,B 0,C 180,E1 11753.075,E2 11753.075} C_VEL
LIN {X 0,Y 368.643,Z 1061.759,A -85,B 0,C 180,E1 11750.379,E2 11750.379} C_VEL
LIN {X 0,Y 373.652,Z 1044.075,A -85,B 0,C 180,E1 11748.012,E2 11748.012} C_VEL
LIN {X 0,Y 379.058,Z 1024.243,A -85,B 0,C 180,E1 11745.771,E2 11745.771} C_VEL
LIN {X 0,Y 383.95,Z 1005.054,A -85,B 0,C 180,E1 11743.942,E2 11743.942} C_VEL
LIN {X 0,Y 388.588,Z 984.758,A -85,B 0,C 180,E1 11742.338,E2 11742.338} C_VEL
LIN {X 0,Y 392.877,Z 964.046,A -85,B 0,C 180,E1 11740.975,E2 11740.975} C_VEL
LIN {X 0,Y 396.616,Z 942.479,A -85,B 0,C 180,E1 11739.846,E2 11739.846} C_VEL
LIN {X 0,Y 400.048,Z 918.526,A -85,B 0,C 180,E1 11738.872,E2 11738.872} C_VEL
LIN {X 0,Y 402.535,Z 895.882,A -85,B 0,C 180,E1 11738.203,E2 11738.203} C_VEL
LIN {X 0,Y 404.782,Z 858.025,A -85,B 0,C 180,E1 11737.408,E2 11737.408} C_VEL
LIN {X 0,Y 415.744,Z 650.399,A -85,B 0,C 180,E1 11733.291,E2 11733.291} C_VEL
LIN {X 0,Y 416.475,Z 635.402,A -85,B 0,C 180,E1 11732.981,E2 11732.981} C_VEL
LIN {X 0,Y 406.45,Z 619.859,A -85,B 0,C 180,E1 11730.447,E2 11730.447} C_VEL
LIN {X 0,Y 396.91,Z 606.23,A -85,B 0,C 180,E1 11727.777,E2 11727.777} C_VEL
LIN {X 0,Y 388.751,Z 595.406,A -85,B 0,C 180,E1 11725.233,E2 11725.233} C_VEL
LIN {X 0,Y 384.372,Z 589.84,A -85,B 0,C 180,E1 11723.737,E2 11723.737} C_VEL
LIN {X 0,Y 380.483,Z 585.046,A -85,B 0,C 180,E1 11722.316,E2 11722.316} C_VEL
LIN {X 0,Y 376.715,Z 580.416,A -85,B 0,C 180,E1 11720.833,E2 11720.833} C_VEL
LIN {X 0,Y 372.336,Z 575.26,A -85,B 0,C 180,E1 11718.961,E2 11718.961} C_VEL
LIN {X 0,Y 367.269,Z 569.496,A -85,B 0,C 180,E1 11716.528,E2 11716.528} C_VEL
LIN {X 0,Y 362.038,Z 563.674,A -85,B 0,C 180,E1 11713.576,E2 11713.576} C_VEL
LIN {X 0,Y 358.857,Z 560.54,A -85,B 0,C 180,E1 11711.246,E2 11711.246} C_VEL
LIN {X 0,Y 357.684,Z 557.772,A -85,B 0,C 180,E1 11709.168,E2 11709.168} C_VEL
LIN {X 0,Y 354.549,Z 553.432,A -85,B 0,C 180,E1 11701.777,E2 11701.777} C_VEL
LIN {X 0,Y 354.362,Z 552.854,A -85,B 0,C 180,E1 11698.221,E2 11698.221} C_VEL
LIN {X 0,Y 354.754,Z 554.055,A -85,B 0,C 180,E1 11694.338,E2 11694.338} C_VEL
LIN {X 0,Y 357.89,Z 558.157,A -85,B 0,C 180,E1 11687.905,E2 11687.905} C_VEL
LIN {X 0,Y 360.355,Z 562.652,A -85,B 0,C 180,E1 11684.386,E2 11684.386} C_VEL
LIN {X 0,Y 361.297,Z 563.806,A -85,B 0,C 180,E1 11683.438,E2 11683.438} C_VEL
LIN {X 0,Y 363.691,Z 568.059,A -85,B 0,C 180,E1 11680.903,E2 11680.903} C_VEL
LIN {X 0,Y 364.554,Z 569.443,A -85,B 0,C 180,E1 11680.117,E2 11680.117} C_VEL
LIN {X 0,Y 367.025,Z 573.536,A -85,B 0,C 180,E1 11678.085,E2 11678.085} C_VEL
LIN {X 0,Y 372.958,Z 581.271,A -85,B 0,C 180,E1 11675.235,E2 11675.235} C_VEL
LIN {X 0,Y 377.234,Z 586.945,A -85,B 0,C 180,E1 11673.431,E2 11673.431} C_VEL
LIN {X 0,Y 380.616,Z 591.347,A -85,B 0,C 180,E1 11672.121,E2 11672.121} C_VEL
LIN {X 0,Y 387.733,Z 601.217,A -85,B 0,C 180,E1 11669.597,E2 11669.597} C_VEL
LIN {X 0,Y 395.572,Z 612.381,A -85,B 0,C 180,E1 11667.125,E2 11667.125} C_VEL
LIN {X 0,Y 405.233,Z 627.463,A -85,B 0,C 180,E1 11664.387,E2 11664.387} C_VEL
LIN {X 0,Y 413.486,Z 641.242,A -85,B 0,C 180,E1 11662.272,E2 11662.272} C_VEL
LIN {X 0,Y 402.933,Z 872.594,A -85,B 0,C 180,E1 11657.981,E2 11657.981} C_VEL
LIN {X 0,Y 401.227,Z 902.124,A -85,B 0,C 180,E1 11657.379,E2 11657.379} C_VEL
LIN {X 0,Y 398.898,Z 924.044,A -85,B 0,C 180,E1 11656.732,E2 11656.732} C_VEL
LIN {X 0,Y 395.772,Z 945.242,A -85,B 0,C 180,E1 11655.847,E2 11655.847} C_VEL
LIN {X 0,Y 391.889,Z 966.638,A -85,B 0,C 180,E1 11654.689,E2 11654.689} C_VEL
LIN {X 0,Y 387.844,Z 985.488,A -85,B 0,C 180,E1 11653.418,E2 11653.418} C_VEL
LIN {X 0,Y 383.086,Z 1004.658,A -85,B 0,C 180,E1 11651.825,E2 11651.825} C_VEL
LIN {X 0,Y 378.09,Z 1022.998,A -85,B 0,C 180,E1 11649.987,E2 11649.987} C_VEL
LIN {X 0,Y 373.089,Z 1039.846,A -85,B 0,C 180,E1 11647.956,E2 11647.956} C_VEL
LIN {X 0,Y 367.855,Z 1056.405,A -85,B 0,C 180,E1 11645.568,E2 11645.568} C_VEL
LIN {X 0,Y 363.055,Z 1071.179,A -85,B 0,C 180,E1 11643.045,E2 11643.045} C_VEL
LIN {X 0,Y 358.377,Z 1085.307,A -85,B 0,C 180,E1 11640.145,E2 11640.145} C_VEL
LIN {X 0,Y 354.245,Z 1097.98,A -85,B 0,C 180,E1 11637.028,E2 11637.028} C_VEL
LIN {X 0,Y 350.783,Z 1109.258,A -85,B 0,C 180,E1 11633.697,E2 11633.697} C_VEL
LIN {X 0,Y 348.16,Z 1118.587,A -85,B 0,C 180,E1 11630.334,E2 11630.334} C_VEL
LIN {X 0,Y 346.229,Z 1126.533,A -85,B 0,C 180,E1 11626.785,E2 11626.785} C_VEL
LIN {X 0,Y 345.082,Z 1132.447,A -85,B 0,C 180,E1 11623.507,E2 11623.507} C_VEL
LIN {X 0,Y 343.784,Z 1134.417,A -85,B 0,C 180,E1 11622.277,E2 11622.277} C_VEL
LIN {X 0,Y 336.899,Z 1138.897,A -85,B 0,C 180,E1 11618.865,E2 11618.865} C_VEL
LIN {X 0,Y 336.159,Z 1139.83,A -85,B 0,C 180,E1 11617.841,E2 11617.841} C_VEL
LIN {X 0,Y 335.995,Z 1142.286,A -85,B 0,C 180,E1 11614.096,E2 11614.096} C_VEL
LIN {X 0,Y 335.957,Z 1143.167,A -85,B 0,C 180,E1 11610.682,E2 11610.682} C_VEL
LIN {X 0,Y 335.968,Z 1142.77,A -85,B 0,C 180,E1 11607.1,E2 11607.1} C_VEL
LIN {X 0,Y 336.073,Z 1141.078,A -85,B 0,C 180,E1 11603.68,E2 11603.68} C_VEL
LIN {X 0,Y 336.398,Z 1137.725,A -85,B 0,C 180,E1 11599.9,E2 11599.9} C_VEL
LIN {X 0,Y 337.139,Z 1133.058,A -85,B 0,C 180,E1 11596.275,E2 11596.275} C_VEL
LIN {X 0,Y 338.514,Z 1126.543,A -85,B 0,C 180,E1 11592.562,E2 11592.562} C_VEL
LIN {X 0,Y 340.81,Z 1117.832,A -85,B 0,C 180,E1 11588.667,E2 11588.667} C_VEL
LIN {X 0,Y 343.812,Z 1108.049,A -85,B 0,C 180,E1 11585.141,E2 11585.141} C_VEL
LIN {X 0,Y 347.498,Z 1096.814,A -85,B 0,C 180,E1 11581.844,E2 11581.844} C_VEL
LIN {X 0,Y 351.969,Z 1083.829,A -85,B 0,C 180,E1 11578.677,E2 11578.677} C_VEL
LIN {X 0,Y 356.709,Z 1070.304,A -85,B 0,C 180,E1 11575.902,E2 11575.902} C_VEL
LIN {X 0,Y 361.799,Z 1055.344,A -85,B 0,C 180,E1 11573.349,E2 11573.349} C_VEL
LIN {X 0,Y 367.498,Z 1037.93,A -85,B 0,C 180,E1 11570.86,E2 11570.86} C_VEL
LIN {X 0,Y 372.747,Z 1020.999,A -85,B 0,C 180,E1 11568.837,E2 11568.837} C_VEL
LIN {X 0,Y 377.836,Z 1002.812,A -85,B 0,C 180,E1 11567.045,E2 11567.045} C_VEL
LIN {X 0,Y 382.965,Z 982.373,A -85,B 0,C 180,E1 11565.387,E2 11565.387} C_VEL
LIN {X 0,Y 387.205,Z 963.173,A -85,B 0,C 180,E1 11564.121,E2 11564.121} C_VEL
LIN {X 0,Y 390.901,Z 942.656,A -85,B 0,C 180,E1 11563.052,E2 11563.052} C_VEL
LIN {X 0,Y 394.174,Z 920.218,A -85,B 0,C 180,E1 11562.163,E2 11562.163} C_VEL
LIN {X 0,Y 396.52,Z 898.253,A -85,B 0,C 180,E1 11561.543,E2 11561.543} C_VEL
LIN {X 0,Y 399.094,Z 846.328,A -85,B 0,C 180,E1 11560.545,E2 11560.545} C_VEL
LIN {X 0,Y 406.358,Z 691.996,A -85,B 0,C 180,E1 11557.654,E2 11557.654} C_VEL
LIN {X 0,Y 399.412,Z 702.412,A -85,B 0,C 180,E1 11556.529,E2 11556.529} C_VEL
LIN {X 0,Y 394.555,Z 708.217,A -85,B 0,C 180,E1 11555.652,E2 11555.652} C_VEL
LIN {X 0,Y 389.159,Z 717.261,A -85,B 0,C 180,E1 11554.71,E2 11554.71} C_VEL
LIN {X 0,Y 384.58,Z 722.969,A -85,B 0,C 180,E1 11553.806,E2 11553.806} C_VEL
LIN {X 0,Y 383.421,Z 724.866,A -85,B 0,C 180,E1 11553.585,E2 11553.585} C_VEL
LIN {X 0,Y 378.423,Z 734.134,A -85,B 0,C 180,E1 11552.639,E2 11552.639} C_VEL
LIN {X 0,Y 374.846,Z 739.45,A -85,B 0,C 180,E1 11551.88,E2 11551.88} C_VEL
LIN {X 0,Y 370.084,Z 760.469,A -85,B 0,C 180,E1 11551.349,E2 11551.349} C_VEL
LIN {X 0,Y 366.768,Z 771.928,A -85,B 0,C 180,E1 11550.844,E2 11550.844} C_VEL
LIN {X 0,Y 364.437,Z 778.533,A -85,B 0,C 180,E1 11550.422,E2 11550.422} C_VEL
LIN {X 0,Y 357.624,Z 809.813,A -85,B 0,C 180,E1 11549.62,E2 11549.62} C_VEL
LIN {X 0,Y 354.556,Z 820.987,A -85,B 0,C 180,E1 11549.12,E2 11549.12} C_VEL
LIN {X 0,Y 352.507,Z 827.784,A -85,B 0,C 180,E1 11548.609,E2 11548.609} C_VEL
LIN {X 0,Y 351.752,Z 837.614,A -85,B 0,C 180,E1 11548.24,E2 11548.24} C_VEL
LIN {X 0,Y 349.779,Z 904.591,A -85,B 0,C 180,E1 11546.535,E2 11546.535} C_VEL
LIN {X 0,Y 349.067,Z 923.03,A -85,B 0,C 180,E1 11545.748,E2 11545.748} C_VEL
LIN {X 0,Y 348.069,Z 940.423,A -85,B 0,C 180,E1 11544.706,E2 11544.706} C_VEL
LIN {X 0,Y 346.865,Z 956.525,A -85,B 0,C 180,E1 11543.441,E2 11543.441} C_VEL
LIN {X 0,Y 345.45,Z 972.541,A -85,B 0,C 180,E1 11541.835,E2 11541.835} C_VEL
LIN {X 0,Y 343.962,Z 987.501,A -85,B 0,C 180,E1 11539.972,E2 11539.972} C_VEL
LIN {X 0,Y 342.488,Z 1001.141,A -85,B 0,C 180,E1 11537.851,E2 11537.851} C_VEL
LIN {X 0,Y 341.227,Z 1012.736,A -85,B 0,C 180,E1 11535.64,E2 11535.64} C_VEL
LIN {X 0,Y 340.171,Z 1022.875,A -85,B 0,C 180,E1 11533.254,E2 11533.254} C_VEL
LIN {X 0,Y 339.332,Z 1031.505,A -85,B 0,C 180,E1 11530.698,E2 11530.698} C_VEL
LIN {X 0,Y 338.77,Z 1038.663,A -85,B 0,C 180,E1 11527.974,E2 11527.974} C_VEL
LIN {X 0,Y 338.482,Z 1043.871,A -85,B 0,C 180,E1 11525.255,E2 11525.255} C_VEL
LIN {X 0,Y 338.423,Z 1047.323,A -85,B 0,C 180,E1 11522.54,E2 11522.54} C_VEL
LIN {X 0,Y 338.568,Z 1049.229,A -85,B 0,C 180,E1 11519.662,E2 11519.662} C_VEL
LIN {X 0,Y 338.86,Z 1049.311,A -85,B 0,C 180,E1 11516.956,E2 11516.956} C_VEL
LIN {X 0,Y 339.346,Z 1047.697,A -85,B 0,C 180,E1 11514.251,E2 11514.251} C_VEL
LIN {X 0,Y 340.092,Z 1044.37,A -85,B 0,C 180,E1 11511.547,E2 11511.547} C_VEL
LIN {X 0,Y 341.143,Z 1039.209,A -85,B 0,C 180,E1 11508.847,E2 11508.847} C_VEL
LIN {X 0,Y 342.399,Z 1032.377,A -85,B 0,C 180,E1 11506.319,E2 11506.319} C_VEL
LIN {X 0,Y 343.949,Z 1023.422,A -85,B 0,C 180,E1 11503.796,E2 11503.796} C_VEL
LIN {X 0,Y 345.538,Z 1013.484,A -85,B 0,C 180,E1 11501.615,E2 11501.615} C_VEL
LIN {X 0,Y 347.326,Z 1000.933,A -85,B 0,C 180,E1 11499.44,E2 11499.44} C_VEL
LIN {X 0,Y 348.891,Z 988.284,A -85,B 0,C 180,E1 11497.688,E2 11497.688} C_VEL
LIN {X 0,Y 350.43,Z 973.037,A -85,B 0,C 180,E1 11496.01,E2 11496.01} C_VEL
LIN {X 0,Y 351.67,Z 957.566,A -85,B 0,C 180,E1 11494.675,E2 11494.675} C_VEL
LIN {X 0,Y 352.681,Z 940.132,A -85,B 0,C 180,E1 11493.526,E2 11493.526} C_VEL
LIN {X 0,Y 353.288,Z 922.702,A -85,B 0,C 180,E1 11492.696,E2 11492.696} C_VEL
LIN {X 0,Y 353.949,Z 903.221,A -85,B 0,C 180,E1 11491.99,E2 11491.99} C_VEL
LIN {X 0,Y 355.08,Z 899.549,A -85,B 0,C 180,E1 11491.698,E2 11491.698} C_VEL
LIN {X 0,Y 357.782,Z 893.782,A -85,B 0,C 180,E1 11491.283,E2 11491.283} C_VEL
LIN {X 0,Y 361.428,Z 882.104,A -85,B 0,C 180,E1 11490.864,E2 11490.864} C_VEL
LIN {X 0,Y 366.147,Z 863.482,A -85,B 0,C 180,E1 11490.379,E2 11490.379} C_VEL
LIN {X 0,Y 370.344,Z 852.23,A -85,B 0,C 180,E1 11489.762,E2 11489.762} C_VEL
LIN {X 0,Y 375.249,Z 834.956,A -85,B 0,C 180,E1 11489.22,E2 11489.22} C_VEL
LIN {X 0,Y 379.245,Z 819.542,A -85,B 0,C 180,E1 11488.842,E2 11488.842} C_VEL
LIN {X 0,Y 383.274,Z 809.089,A -85,B 0,C 180,E1 11488.3,E2 11488.3} C_VEL
LIN {X 0,Y 388.262,Z 792.178,A -85,B 0,C 180,E1 11487.787,E2 11487.787} C_VEL
LIN {X 0,Y 392.487,Z 776.266,A -85,B 0,C 180,E1 11487.421,E2 11487.421} C_VEL
LIN {X 0,Y 397.068,Z 764.249,A -85,B 0,C 180,E1 11486.868,E2 11486.868} C_VEL
LIN {X 0,Y 400.729,Z 755.674,A -85,B 0,C 180,E1 11486.408,E2 11486.408} C_VEL
LIN {X 0,Y 402.009,Z 753.346,A -85,B 0,C 180,E1 11486.229,E2 11486.229} C_VEL
LIN {X 0,Y 405.646,Z 749.145,A -85,B 0,C 180,E1 11485.659,E2 11485.659} C_VEL
LIN {X 0,Y 397.752,Z 891.92,A -85,B 0,C 180,E1 11482.776,E2 11482.776} C_VEL
LIN {X 0,Y 395.262,Z 915.362,A -85,B 0,C 180,E1 11482.115,E2 11482.115} C_VEL
LIN {X 0,Y 392.189,Z 937.376,A -85,B 0,C 180,E1 11481.272,E2 11481.272} C_VEL
LIN {X 0,Y 388.434,Z 958.567,A -85,B 0,C 180,E1 11480.207,E2 11480.207} C_VEL
LIN {X 0,Y 383.879,Z 980.666,A -85,B 0,C 180,E1 11478.828,E2 11478.828} C_VEL
LIN {X 0,Y 379.112,Z 1000.972,A -85,B 0,C 180,E1 11477.266,E2 11477.266} C_VEL
LIN {X 0,Y 373.778,Z 1021.434,A -85,B 0,C 180,E1 11475.362,E2 11475.362} C_VEL
LIN {X 0,Y 368.464,Z 1040.526,A -85,B 0,C 180,E1 11473.25,E2 11473.25} C_VEL
LIN {X 0,Y 363.092,Z 1058.391,A -85,B 0,C 180,E1 11470.887,E2 11470.887} C_VEL
LIN {X 0,Y 357.615,Z 1076.306,A -85,B 0,C 180,E1 11468.094,E2 11468.094} C_VEL
LIN {X 0,Y 352.931,Z 1091.495,A -85,B 0,C 180,E1 11465.306,E2 11465.306} C_VEL
LIN {X 0,Y 348.392,Z 1106.425,A -85,B 0,C 180,E1 11462.069,E2 11462.069} C_VEL
LIN {X 0,Y 344.682,Z 1119.372,A -85,B 0,C 180,E1 11458.786,E2 11458.786} C_VEL
LIN {X 0,Y 341.567,Z 1131.027,A -85,B 0,C 180,E1 11455.242,E2 11455.242} C_VEL
LIN {X 0,Y 339.141,Z 1141.504,A -85,B 0,C 180,E1 11451.443,E2 11451.443} C_VEL
LIN {X 0,Y 337.684,Z 1149.081,A -85,B 0,C 180,E1 11448.112,E2 11448.112} C_VEL
LIN {X 0,Y 336.645,Z 1156.15,A -85,B 0,C 180,E1 11444.272,E2 11444.272} C_VEL
LIN {X 0,Y 336.189,Z 1160.825,A -85,B 0,C 180,E1 11440.973,E2 11440.973} C_VEL
LIN {X 0,Y 335.954,Z 1164.747,A -85,B 0,C 180,E1 11437.181,E2 11437.181} C_VEL
LIN {X 0,Y 335.935,Z 1166.811,A -85,B 0,C 180,E1 11433.754,E2 11433.754} C_VEL
LIN {X 0,Y 335.931,Z 1167.623,A -85,B 0,C 180,E1 11430.512,E2 11430.512} C_VEL
LIN {X 0,Y 335.923,Z 1167.098,A -85,B 0,C 180,E1 11426.929,E2 11426.929} C_VEL
LIN {X 0,Y 335.957,Z 1165.35,A -85,B 0,C 180,E1 11423.678,E2 11423.678} C_VEL
LIN {X 0,Y 336.09,Z 1162.006,A -85,B 0,C 180,E1 11419.966,E2 11419.966} C_VEL
LIN {X 0,Y 336.517,Z 1157.222,A -85,B 0,C 180,E1 11416.425,E2 11416.425} C_VEL
LIN {X 0,Y 337.406,Z 1150.903,A -85,B 0,C 180,E1 11412.762,E2 11412.762} C_VEL
LIN {X 0,Y 338.871,Z 1142.773,A -85,B 0,C 180,E1 11409.083,E2 11409.083} C_VEL
LIN {X 0,Y 341.092,Z 1133,A -85,B 0,C 180,E1 11405.402,E2 11405.402} C_VEL
LIN {X 0,Y 343.994,Z 1121.755,A -85,B 0,C 180,E1 11401.909,E2 11401.909} C_VEL
LIN {X 0,Y 347.973,Z 1107.83,A -85,B 0,C 180,E1 11398.267,E2 11398.267} C_VEL
LIN {X 0,Y 352.41,Z 1093.211,A -85,B 0,C 180,E1 11395.032,E2 11395.032} C_VEL
LIN {X 0,Y 357.221,Z 1077.515,A -85,B 0,C 180,E1 11392.121,E2 11392.121} C_VEL
LIN {X 0,Y 362.695,Z 1059.648,A -85,B 0,C 180,E1 11389.297,E2 11389.297} C_VEL
LIN {X 0,Y 367.894,Z 1042.285,A -85,B 0,C 180,E1 11386.977,E2 11386.977} C_VEL
LIN {X 0,Y 373.362,Z 1022.858,A -85,B 0,C 180,E1 11384.792,E2 11384.792} C_VEL
LIN {X 0,Y 378.46,Z 1003.624,A -85,B 0,C 180,E1 11382.961,E2 11382.961} C_VEL
LIN {X 0,Y 383.398,Z 982.6,A -85,B 0,C 180,E1 11381.316,E2 11381.316} C_VEL
LIN {X 0,Y 388.173,Z 959.715,A -85,B 0,C 180,E1 11379.862,E2 11379.862} C_VEL
LIN {X 0,Y 392.044,Z 937.944,A -85,B 0,C 180,E1 11378.76,E2 11378.76} C_VEL
LIN {X 0,Y 395.157,Z 915.801,A -85,B 0,C 180,E1 11377.905,E2 11377.905} C_VEL
LIN {X 0,Y 397.668,Z 892.443,A -85,B 0,C 180,E1 11377.241,E2 11377.241} C_VEL
LIN {X 0,Y 404.188,Z 774.868,A -85,B 0,C 180,E1 11374.86,E2 11374.86} C_VEL
LIN {X 0,Y 411.656,Z 639.547,A -85,B 0,C 180,E1 11372.161,E2 11372.161} C_VEL
LIN {X 0,Y 402.602,Z 625.393,A -85,B 0,C 180,E1 11369.781,E2 11369.781} C_VEL
LIN {X 0,Y 393.808,Z 612.662,A -85,B 0,C 180,E1 11367.235,E2 11367.235} C_VEL
LIN {X 0,Y 386.018,Z 602.142,A -85,B 0,C 180,E1 11364.728,E2 11364.728} C_VEL
LIN {X 0,Y 379.584,Z 593.743,A -85,B 0,C 180,E1 11362.413,E2 11362.413} C_VEL
LIN {X 0,Y 374.153,Z 587.176,A -85,B 0,C 180,E1 11360.246,E2 11360.246} C_VEL
LIN {X 0,Y 370.372,Z 582.634,A -85,B 0,C 180,E1 11358.575,E2 11358.575} C_VEL
LIN {X 0,Y 365.554,Z 577.043,A -85,B 0,C 180,E1 11356.199,E2 11356.199} C_VEL
LIN {X 0,Y 360.555,Z 571.367,A -85,B 0,C 180,E1 11353.306,E2 11353.306} C_VEL
LIN {X 0,Y 355.386,Z 565.858,A -85,B 0,C 180,E1 11349.554,E2 11349.554} C_VEL
LIN {X 0,Y 351.889,Z 562.746,A -85,B 0,C 180,E1 11345.871,E2 11345.871} C_VEL
LIN {X 0,Y 350.709,Z 560.23,A -85,B 0,C 180,E1 11340.98,E2 11340.98} C_VEL
LIN {X 0,Y 350.625,Z 560.009,A -85,B 0,C 180,E1 11337.548,E2 11337.548} C_VEL
LIN {X 0,Y 351.143,Z 561.533,A -85,B 0,C 180,E1 11333.597,E2 11333.597} C_VEL
LIN {X 0,Y 353.945,Z 565.014,A -85,B 0,C 180,E1 11328.099,E2 11328.099} C_VEL
LIN {X 0,Y 356.331,Z 569.517,A -85,B 0,C 180,E1 11324.539,E2 11324.539} C_VEL
LIN {X 0,Y 357.278,Z 570.712,A -85,B 0,C 180,E1 11323.581,E2 11323.581} C_VEL
LIN {X 0,Y 360.554,Z 575.277,A -85,B 0,C 180,E1 11321.151,E2 11321.151} C_VEL
LIN {X 0,Y 361.931,Z 577.004,A -85,B 0,C 180,E1 11320.303,E2 11320.303} C_VEL
